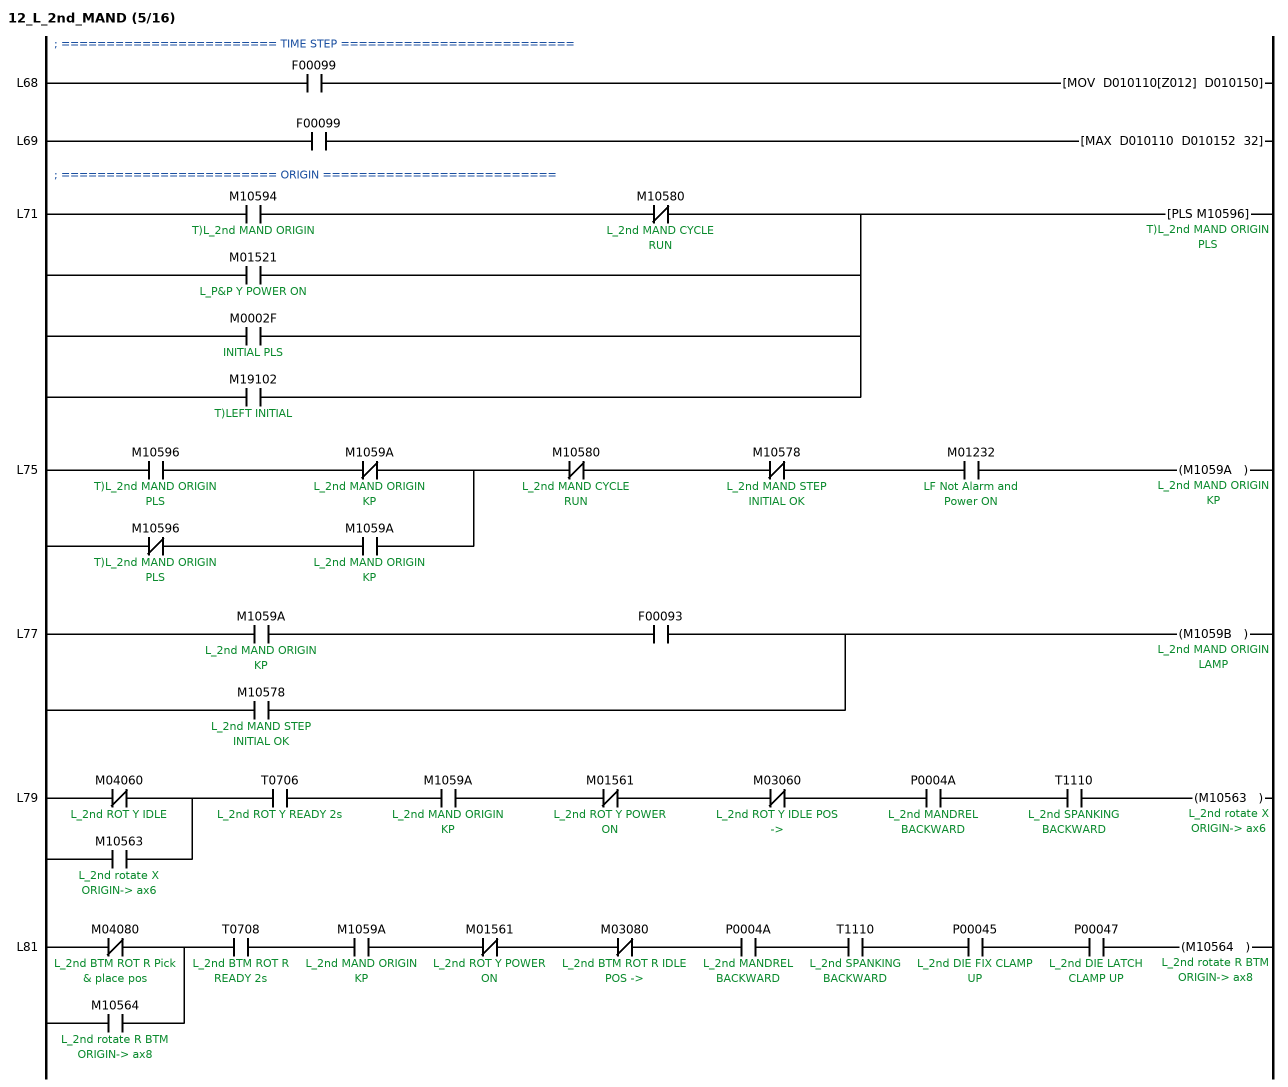
[picture p72: 12_L_2nd_MAND rungs L68-L81]
// ======================== TIME STEP ==========================
; L68
LOAD      F00099
MOV       D010110[Z012] D010150
; L69
LOAD      F00099
MAX       D010110 D010152 32
// ======================== ORIGIN ==========================
; L71
LOAD      M10594	// T)L_2nd MAND ORIGIN
AND NOT   M10580	// L_2nd MAND CYCLE RUN
OR        M01521	// L_P&P Y POWER ON
OR        M0002F	// INITIAL PLS
OR        M19102	// T)LEFT INITIAL
OUTP      M10596	// T)L_2nd MAND ORIGIN PLS
; L75
LOAD      M10596	// T)L_2nd MAND ORIGIN PLS
AND NOT   M1059A	// L_2nd MAND ORIGIN KP
LOAD NOT  M10596	// T)L_2nd MAND ORIGIN PLS
AND       M1059A	// L_2nd MAND ORIGIN KP
OR LOAD
AND NOT   M10580	// L_2nd MAND CYCLE RUN
AND NOT   M10578	// L_2nd MAND STEP INITIAL OK
AND       M01232	// LF Not Alarm and Power ON
OUT       M1059A	// L_2nd MAND ORIGIN KP
; L77
LOAD      M1059A	// L_2nd MAND ORIGIN KP
AND       F00093
OR        M10578	// L_2nd MAND STEP INITIAL OK
OUT       M1059B	// L_2nd MAND ORIGIN LAMP
; L79
LOAD NOT  M04060	// L_2nd ROT Y IDLE
OR        M10563	// L_2nd rotate X ORIGIN-> ax6
AND       T0706	// L_2nd ROT Y READY 2s
AND       M1059A	// L_2nd MAND ORIGIN KP
AND NOT   M01561	// L_2nd ROT Y POWER ON
AND NOT   M03060	// L_2nd ROT Y IDLE POS ->
AND       P0004A	// L_2nd MANDREL BACKWARD
AND       T1110	// L_2nd SPANKING BACKWARD
OUT       M10563	// L_2nd rotate X ORIGIN-> ax6
; L81
LOAD NOT  M04080	// L_2nd BTM ROT R Pick & place pos
OR        M10564	// L_2nd rotate R BTM  ORIGIN-> ax8
AND       T0708	// L_2nd BTM ROT R READY 2s
AND       M1059A	// L_2nd MAND ORIGIN KP
AND NOT   M01561	// L_2nd ROT Y POWER ON
AND NOT   M03080	// L_2nd BTM ROT R IDLE POS ->
AND       P0004A	// L_2nd MANDREL BACKWARD
AND       T1110	// L_2nd SPANKING BACKWARD
AND       P00045	// L_2nd DIE FIX CLAMP UP
AND       P00047	// L_2nd DIE LATCH CLAMP UP
OUT       M10564	// L_2nd rotate R BTM  ORIGIN-> ax8

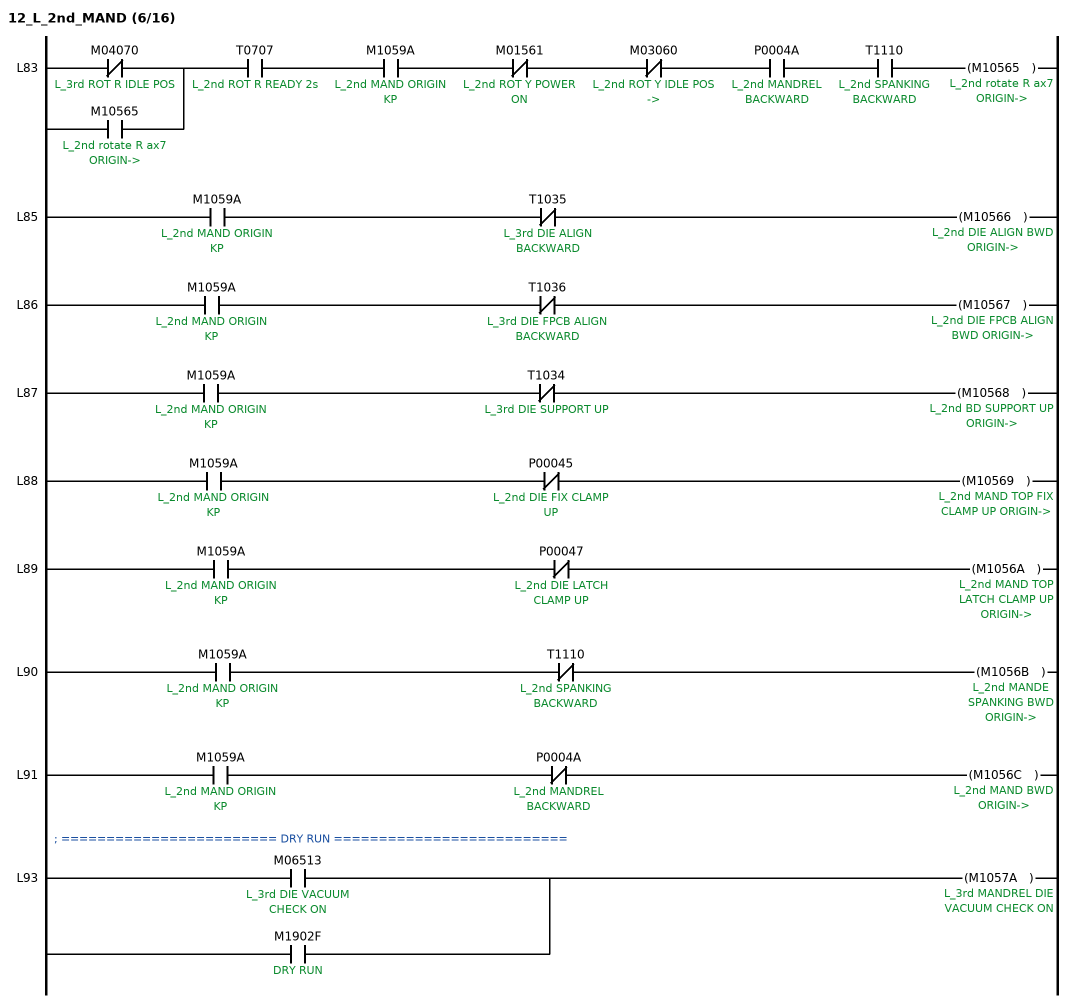
; L83
LOAD NOT  M04070	// L_3rd ROT R IDLE POS
OR        M10565	// L_2nd rotate R ax7 ORIGIN->
AND       T0707	// L_2nd ROT R READY 2s
AND       M1059A	// L_2nd MAND ORIGIN KP
AND NOT   M01561	// L_2nd ROT Y POWER ON
AND NOT   M03060	// L_2nd ROT Y IDLE POS ->
AND       P0004A	// L_2nd MANDREL BACKWARD
AND       T1110	// L_2nd SPANKING BACKWARD
OUT       M10565	// L_2nd rotate R ax7 ORIGIN->
; L85
LOAD      M1059A	// L_2nd MAND ORIGIN KP
AND NOT   T1035	// L_3rd DIE ALIGN BACKWARD
OUT       M10566	// L_2nd DIE ALIGN BWD ORIGIN->
; L86
LOAD      M1059A	// L_2nd MAND ORIGIN KP
AND NOT   T1036	// L_3rd DIE FPCB ALIGN BACKWARD
OUT       M10567	// L_2nd DIE FPCB ALIGN BWD ORIGIN->
; L87
LOAD      M1059A	// L_2nd MAND ORIGIN KP
AND NOT   T1034	// L_3rd DIE SUPPORT UP
OUT       M10568	// L_2nd BD SUPPORT UP ORIGIN->
; L88
LOAD      M1059A	// L_2nd MAND ORIGIN KP
AND NOT   P00045	// L_2nd DIE FIX CLAMP UP
OUT       M10569	// L_2nd MAND TOP FIX CLAMP UP ORIGIN->
; L89
LOAD      M1059A	// L_2nd MAND ORIGIN KP
AND NOT   P00047	// L_2nd DIE LATCH CLAMP UP
OUT       M1056A	// L_2nd MAND TOP LATCH CLAMP UP ORIGIN->
; L90
LOAD      M1059A	// L_2nd MAND ORIGIN KP
AND NOT   T1110	// L_2nd SPANKING BACKWARD
OUT       M1056B	// L_2nd MANDE SPANKING BWD ORIGIN->
; L91
LOAD      M1059A	// L_2nd MAND ORIGIN KP
AND NOT   P0004A	// L_2nd MANDREL BACKWARD
OUT       M1056C	// L_2nd MAND BWD ORIGIN->
// ======================== DRY RUN ==========================
; L93
LOAD      M06513	// L_3rd DIE VACUUM CHECK ON
OR        M1902F	// DRY RUN
OUT       M1057A	// L_3rd MANDREL DIE VACUUM CHECK ON

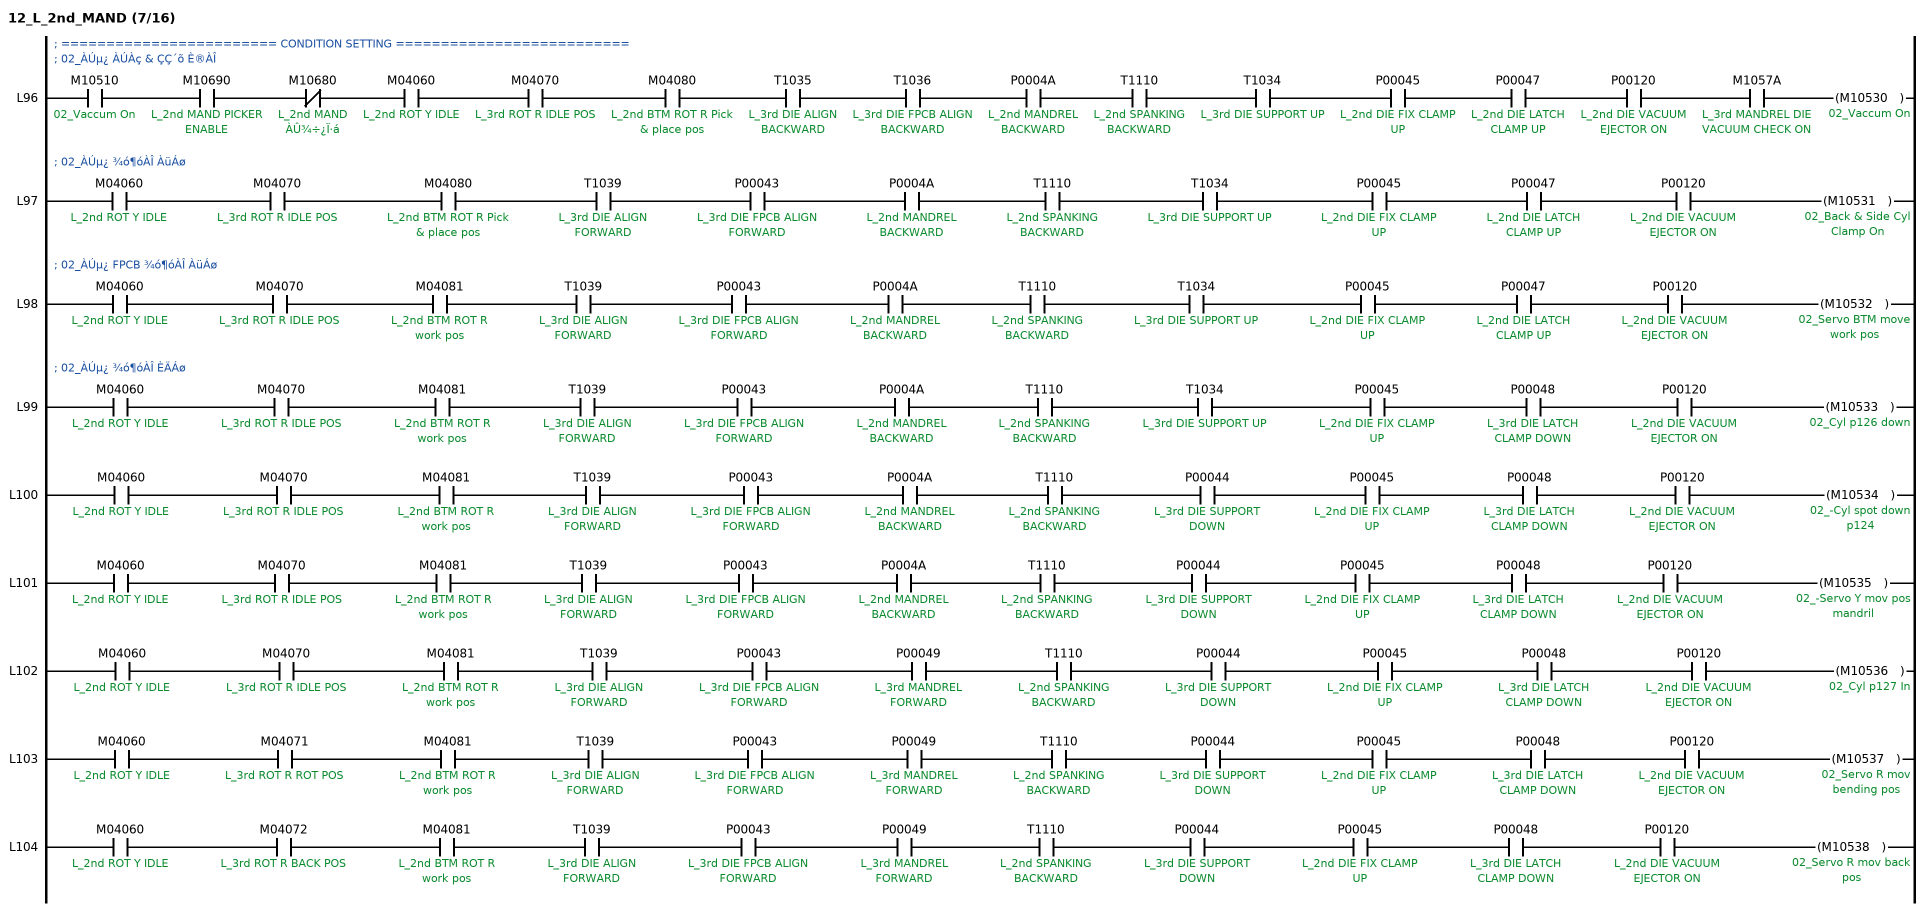
// ======================== CONDITION SETTING ==========================
; L96
LOAD      M10510	// 02_Vaccum On
AND       M10690	// L_2nd MAND PICKER ENABLE
AND NOT   M10680	// L_2nd MAND ÀÛ¾÷¿Ï·á
AND       M04060	// L_2nd ROT Y IDLE
AND       M04070	// L_3rd ROT R IDLE POS
AND       M04080	// L_2nd BTM ROT R Pick & place pos
AND       T1035	// L_3rd DIE ALIGN BACKWARD
AND       T1036	// L_3rd DIE FPCB ALIGN BACKWARD
AND       P0004A	// L_2nd MANDREL BACKWARD
AND       T1110	// L_2nd SPANKING BACKWARD
AND       T1034	// L_3rd DIE SUPPORT UP
AND       P00045	// L_2nd DIE FIX CLAMP UP
AND       P00047	// L_2nd DIE LATCH CLAMP UP
AND       P00120	// L_2nd DIE VACUUM EJECTOR ON
AND       M1057A	// L_3rd MANDREL DIE VACUUM CHECK ON
OUT       M10530	// 02_Vaccum On
// output comment: 02_ÀÚµ¿ ÀÚÀç & ÇÇ´õ È®ÀÎ
; L97
LOAD      M04060	// L_2nd ROT Y IDLE
AND       M04070	// L_3rd ROT R IDLE POS
AND       M04080	// L_2nd BTM ROT R Pick & place pos
AND       T1039	// L_3rd DIE ALIGN FORWARD
AND       P00043	// L_3rd DIE FPCB ALIGN FORWARD
AND       P0004A	// L_2nd MANDREL BACKWARD
AND       T1110	// L_2nd SPANKING BACKWARD
AND       T1034	// L_3rd DIE SUPPORT UP
AND       P00045	// L_2nd DIE FIX CLAMP UP
AND       P00047	// L_2nd DIE LATCH CLAMP UP
AND       P00120	// L_2nd DIE VACUUM EJECTOR ON
OUT       M10531	// 02_Back & Side Cyl Clamp On
// output comment: 02_ÀÚµ¿ ¾ó¶óÀÎ ÀüÁø
; L98
LOAD      M04060	// L_2nd ROT Y IDLE
AND       M04070	// L_3rd ROT R IDLE POS
AND       M04081	// L_2nd BTM ROT R work pos
AND       T1039	// L_3rd DIE ALIGN FORWARD
AND       P00043	// L_3rd DIE FPCB ALIGN FORWARD
AND       P0004A	// L_2nd MANDREL BACKWARD
AND       T1110	// L_2nd SPANKING BACKWARD
AND       T1034	// L_3rd DIE SUPPORT UP
AND       P00045	// L_2nd DIE FIX CLAMP UP
AND       P00047	// L_2nd DIE LATCH CLAMP UP
AND       P00120	// L_2nd DIE VACUUM EJECTOR ON
OUT       M10532	// 02_Servo BTM move work pos
// output comment: 02_ÀÚµ¿ FPCB ¾ó¶óÀÎ ÀüÁø
; L99
LOAD      M04060	// L_2nd ROT Y IDLE
AND       M04070	// L_3rd ROT R IDLE POS
AND       M04081	// L_2nd BTM ROT R work pos
AND       T1039	// L_3rd DIE ALIGN FORWARD
AND       P00043	// L_3rd DIE FPCB ALIGN FORWARD
AND       P0004A	// L_2nd MANDREL BACKWARD
AND       T1110	// L_2nd SPANKING BACKWARD
AND       T1034	// L_3rd DIE SUPPORT UP
AND       P00045	// L_2nd DIE FIX CLAMP UP
AND       P00048	// L_3rd DIE LATCH CLAMP DOWN
AND       P00120	// L_2nd DIE VACUUM EJECTOR ON
OUT       M10533	// 02_Cyl p126 down
// output comment: 02_ÀÚµ¿ ¾ó¶óÀÎ ÈÄÁø
; L100
LOAD      M04060	// L_2nd ROT Y IDLE
AND       M04070	// L_3rd ROT R IDLE POS
AND       M04081	// L_2nd BTM ROT R work pos
AND       T1039	// L_3rd DIE ALIGN FORWARD
AND       P00043	// L_3rd DIE FPCB ALIGN FORWARD
AND       P0004A	// L_2nd MANDREL BACKWARD
AND       T1110	// L_2nd SPANKING BACKWARD
AND       P00044	// L_3rd DIE SUPPORT DOWN
AND       P00045	// L_2nd DIE FIX CLAMP UP
AND       P00048	// L_3rd DIE LATCH CLAMP DOWN
AND       P00120	// L_2nd DIE VACUUM EJECTOR ON
OUT       M10534	// 02_-Cyl spot down p124
; L101
LOAD      M04060	// L_2nd ROT Y IDLE
AND       M04070	// L_3rd ROT R IDLE POS
AND       M04081	// L_2nd BTM ROT R work pos
AND       T1039	// L_3rd DIE ALIGN FORWARD
AND       P00043	// L_3rd DIE FPCB ALIGN FORWARD
AND       P0004A	// L_2nd MANDREL BACKWARD
AND       T1110	// L_2nd SPANKING BACKWARD
AND       P00044	// L_3rd DIE SUPPORT DOWN
AND       P00045	// L_2nd DIE FIX CLAMP UP
AND       P00048	// L_3rd DIE LATCH CLAMP DOWN
AND       P00120	// L_2nd DIE VACUUM EJECTOR ON
OUT       M10535	// 02_-Servo Y mov pos mandril
; L102
LOAD      M04060	// L_2nd ROT Y IDLE
AND       M04070	// L_3rd ROT R IDLE POS
AND       M04081	// L_2nd BTM ROT R work pos
AND       T1039	// L_3rd DIE ALIGN FORWARD
AND       P00043	// L_3rd DIE FPCB ALIGN FORWARD
AND       P00049	// L_3rd MANDREL FORWARD
AND       T1110	// L_2nd SPANKING BACKWARD
AND       P00044	// L_3rd DIE SUPPORT DOWN
AND       P00045	// L_2nd DIE FIX CLAMP UP
AND       P00048	// L_3rd DIE LATCH CLAMP DOWN
AND       P00120	// L_2nd DIE VACUUM EJECTOR ON
OUT       M10536	// 02_Cyl p127 In
; L103
LOAD      M04060	// L_2nd ROT Y IDLE
AND       M04071	// L_3rd ROT R ROT POS
AND       M04081	// L_2nd BTM ROT R work pos
AND       T1039	// L_3rd DIE ALIGN FORWARD
AND       P00043	// L_3rd DIE FPCB ALIGN FORWARD
AND       P00049	// L_3rd MANDREL FORWARD
AND       T1110	// L_2nd SPANKING BACKWARD
AND       P00044	// L_3rd DIE SUPPORT DOWN
AND       P00045	// L_2nd DIE FIX CLAMP UP
AND       P00048	// L_3rd DIE LATCH CLAMP DOWN
AND       P00120	// L_2nd DIE VACUUM EJECTOR ON
OUT       M10537	// 02_Servo R mov bending pos
; L104
LOAD      M04060	// L_2nd ROT Y IDLE
AND       M04072	// L_3rd ROT R BACK POS
AND       M04081	// L_2nd BTM ROT R work pos
AND       T1039	// L_3rd DIE ALIGN FORWARD
AND       P00043	// L_3rd DIE FPCB ALIGN FORWARD
AND       P00049	// L_3rd MANDREL FORWARD
AND       T1110	// L_2nd SPANKING BACKWARD
AND       P00044	// L_3rd DIE SUPPORT DOWN
AND       P00045	// L_2nd DIE FIX CLAMP UP
AND       P00048	// L_3rd DIE LATCH CLAMP DOWN
AND       P00120	// L_2nd DIE VACUUM EJECTOR ON
OUT       M10538	// 02_Servo R mov back pos

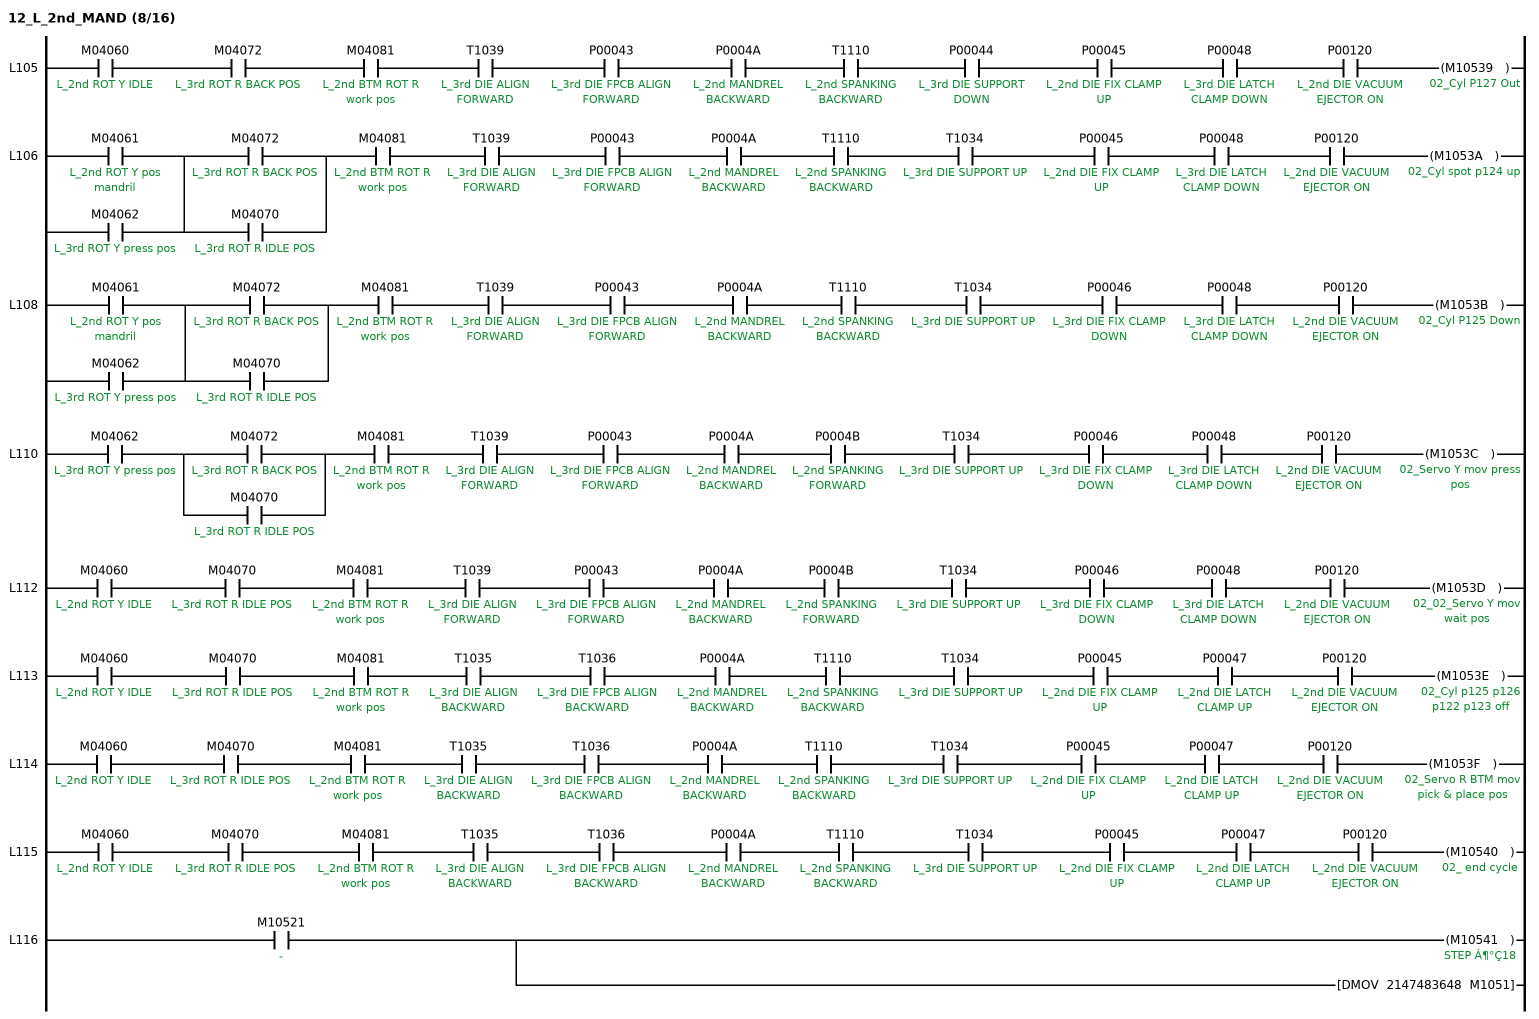
; L105
LOAD      M04060	// L_2nd ROT Y IDLE
AND       M04072	// L_3rd ROT R BACK POS
AND       M04081	// L_2nd BTM ROT R work pos
AND       T1039	// L_3rd DIE ALIGN FORWARD
AND       P00043	// L_3rd DIE FPCB ALIGN FORWARD
AND       P0004A	// L_2nd MANDREL BACKWARD
AND       T1110	// L_2nd SPANKING BACKWARD
AND       P00044	// L_3rd DIE SUPPORT DOWN
AND       P00045	// L_2nd DIE FIX CLAMP UP
AND       P00048	// L_3rd DIE LATCH CLAMP DOWN
AND       P00120	// L_2nd DIE VACUUM EJECTOR ON
OUT       M10539	// 02_Cyl P127 Out
; L106
LOAD      M04061	// L_2nd ROT Y pos mandril
OR        M04062	// L_3rd ROT Y press pos
LOAD      M04072	// L_3rd ROT R BACK POS
OR        M04070	// L_3rd ROT R IDLE POS
AND LOAD
AND       M04081	// L_2nd BTM ROT R work pos
AND       T1039	// L_3rd DIE ALIGN FORWARD
AND       P00043	// L_3rd DIE FPCB ALIGN FORWARD
AND       P0004A	// L_2nd MANDREL BACKWARD
AND       T1110	// L_2nd SPANKING BACKWARD
AND       T1034	// L_3rd DIE SUPPORT UP
AND       P00045	// L_2nd DIE FIX CLAMP UP
AND       P00048	// L_3rd DIE LATCH CLAMP DOWN
AND       P00120	// L_2nd DIE VACUUM EJECTOR ON
OUT       M1053A	// 02_Cyl spot p124 up
; L108
LOAD      M04061	// L_2nd ROT Y pos mandril
OR        M04062	// L_3rd ROT Y press pos
LOAD      M04072	// L_3rd ROT R BACK POS
OR        M04070	// L_3rd ROT R IDLE POS
AND LOAD
AND       M04081	// L_2nd BTM ROT R work pos
AND       T1039	// L_3rd DIE ALIGN FORWARD
AND       P00043	// L_3rd DIE FPCB ALIGN FORWARD
AND       P0004A	// L_2nd MANDREL BACKWARD
AND       T1110	// L_2nd SPANKING BACKWARD
AND       T1034	// L_3rd DIE SUPPORT UP
AND       P00046	// L_3rd DIE FIX CLAMP DOWN
AND       P00048	// L_3rd DIE LATCH CLAMP DOWN
AND       P00120	// L_2nd DIE VACUUM EJECTOR ON
OUT       M1053B	// 02_Cyl P125 Down
; L110
LOAD      M04062	// L_3rd ROT Y press pos
LOAD      M04072	// L_3rd ROT R BACK POS
OR        M04070	// L_3rd ROT R IDLE POS
AND LOAD
AND       M04081	// L_2nd BTM ROT R work pos
AND       T1039	// L_3rd DIE ALIGN FORWARD
AND       P00043	// L_3rd DIE FPCB ALIGN FORWARD
AND       P0004A	// L_2nd MANDREL BACKWARD
AND       P0004B	// L_2nd SPANKING FORWARD
AND       T1034	// L_3rd DIE SUPPORT UP
AND       P00046	// L_3rd DIE FIX CLAMP DOWN
AND       P00048	// L_3rd DIE LATCH CLAMP DOWN
AND       P00120	// L_2nd DIE VACUUM EJECTOR ON
OUT       M1053C	// 02_Servo Y mov press pos
; L112
LOAD      M04060	// L_2nd ROT Y IDLE
AND       M04070	// L_3rd ROT R IDLE POS
AND       M04081	// L_2nd BTM ROT R work pos
AND       T1039	// L_3rd DIE ALIGN FORWARD
AND       P00043	// L_3rd DIE FPCB ALIGN FORWARD
AND       P0004A	// L_2nd MANDREL BACKWARD
AND       P0004B	// L_2nd SPANKING FORWARD
AND       T1034	// L_3rd DIE SUPPORT UP
AND       P00046	// L_3rd DIE FIX CLAMP DOWN
AND       P00048	// L_3rd DIE LATCH CLAMP DOWN
AND       P00120	// L_2nd DIE VACUUM EJECTOR ON
OUT       M1053D	// 02_02_Servo Y mov wait pos
; L113
LOAD      M04060	// L_2nd ROT Y IDLE
AND       M04070	// L_3rd ROT R IDLE POS
AND       M04081	// L_2nd BTM ROT R work pos
AND       T1035	// L_3rd DIE ALIGN BACKWARD
AND       T1036	// L_3rd DIE FPCB ALIGN BACKWARD
AND       P0004A	// L_2nd MANDREL BACKWARD
AND       T1110	// L_2nd SPANKING BACKWARD
AND       T1034	// L_3rd DIE SUPPORT UP
AND       P00045	// L_2nd DIE FIX CLAMP UP
AND       P00047	// L_2nd DIE LATCH CLAMP UP
AND       P00120	// L_2nd DIE VACUUM EJECTOR ON
OUT       M1053E	// 02_Cyl p125 p126 p122 p123 off
; L114
LOAD      M04060	// L_2nd ROT Y IDLE
AND       M04070	// L_3rd ROT R IDLE POS
AND       M04081	// L_2nd BTM ROT R work pos
AND       T1035	// L_3rd DIE ALIGN BACKWARD
AND       T1036	// L_3rd DIE FPCB ALIGN BACKWARD
AND       P0004A	// L_2nd MANDREL BACKWARD
AND       T1110	// L_2nd SPANKING BACKWARD
AND       T1034	// L_3rd DIE SUPPORT UP
AND       P00045	// L_2nd DIE FIX CLAMP UP
AND       P00047	// L_2nd DIE LATCH CLAMP UP
AND       P00120	// L_2nd DIE VACUUM EJECTOR ON
OUT       M1053F	// 02_Servo R BTM mov pick & place pos
; L115
LOAD      M04060	// L_2nd ROT Y IDLE
AND       M04070	// L_3rd ROT R IDLE POS
AND       M04081	// L_2nd BTM ROT R work pos
AND       T1035	// L_3rd DIE ALIGN BACKWARD
AND       T1036	// L_3rd DIE FPCB ALIGN BACKWARD
AND       P0004A	// L_2nd MANDREL BACKWARD
AND       T1110	// L_2nd SPANKING BACKWARD
AND       T1034	// L_3rd DIE SUPPORT UP
AND       P00045	// L_2nd DIE FIX CLAMP UP
AND       P00047	// L_2nd DIE LATCH CLAMP UP
AND       P00120	// L_2nd DIE VACUUM EJECTOR ON
OUT       M10540	// 02_ end cycle
; L116
LOAD      M10521	// -
OUT       M10541	// STEP Á¶°Ç18
DMOV      2147483648 M1051

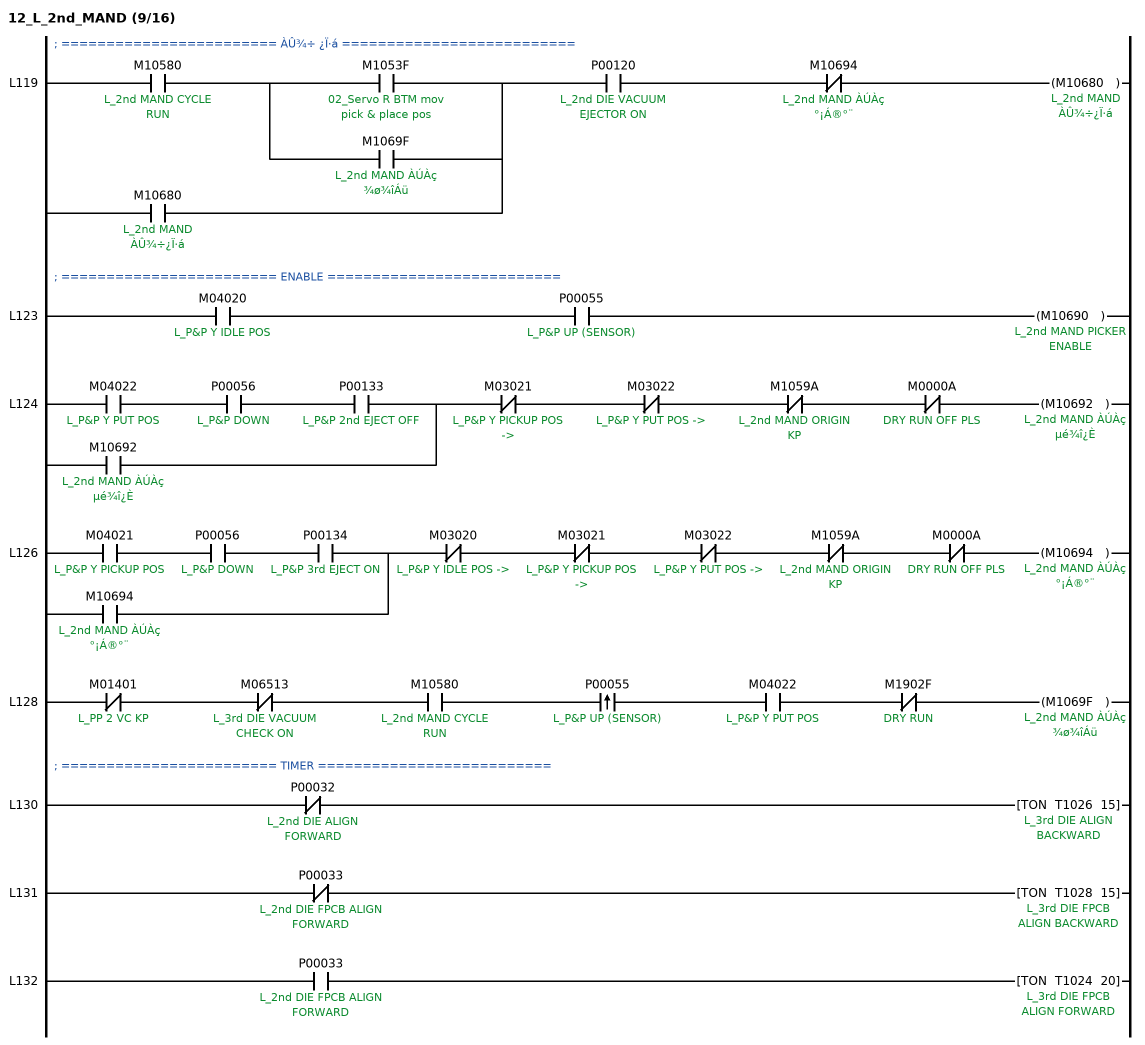
// ======================== ÀÛ¾÷ ¿Ï·á ==========================
; L119
LOAD      M10580	// L_2nd MAND CYCLE RUN
LOAD      M1053F	// 02_Servo R BTM mov pick & place pos
OR        M1069F	// L_2nd MAND ÀÚÀç ¾ø¾îÁü
AND LOAD
OR        M10680	// L_2nd MAND ÀÛ¾÷¿Ï·á
AND       P00120	// L_2nd DIE VACUUM EJECTOR ON
AND NOT   M10694	// L_2nd MAND ÀÚÀç °¡Á®°¨
OUT       M10680	// L_2nd MAND ÀÛ¾÷¿Ï·á
// ======================== ENABLE ==========================
; L123
LOAD      M04020	// L_P&P Y IDLE POS
AND       P00055	// L_P&P UP (SENSOR)
OUT       M10690	// L_2nd MAND PICKER ENABLE
; L124
LOAD      M04022	// L_P&P Y PUT POS
AND       P00056	// L_P&P DOWN
AND       P00133	// L_P&P 2nd EJECT OFF
OR        M10692	// L_2nd MAND ÀÚÀç µé¾î¿È
AND NOT   M03021	// L_P&P Y PICKUP POS ->
AND NOT   M03022	// L_P&P Y PUT POS ->
AND NOT   M1059A	// L_2nd MAND ORIGIN KP
AND NOT   M0000A	// DRY RUN OFF PLS
OUT       M10692	// L_2nd MAND ÀÚÀç µé¾î¿È
; L126
LOAD      M04021	// L_P&P Y PICKUP POS
AND       P00056	// L_P&P DOWN
AND       P00134	// L_P&P 3rd EJECT ON
OR        M10694	// L_2nd MAND ÀÚÀç °¡Á®°¨
AND NOT   M03020	// L_P&P Y IDLE POS ->
AND NOT   M03021	// L_P&P Y PICKUP POS ->
AND NOT   M03022	// L_P&P Y PUT POS ->
AND NOT   M1059A	// L_2nd MAND ORIGIN KP
AND NOT   M0000A	// DRY RUN OFF PLS
OUT       M10694	// L_2nd MAND ÀÚÀç °¡Á®°¨
; L128
LOAD NOT  M01401	// L_PP 2 VC KP
AND NOT   M06513	// L_3rd DIE VACUUM CHECK ON
AND       M10580	// L_2nd MAND CYCLE RUN
ANDP      P00055	// L_P&P UP (SENSOR)
AND       M04022	// L_P&P Y PUT POS
AND NOT   M1902F	// DRY RUN
OUT       M1069F	// L_2nd MAND ÀÚÀç ¾ø¾îÁü
// ======================== TIMER ==========================
; L130
LOAD NOT  P00032	// L_2nd DIE ALIGN FORWARD
TON       T1026 15	// L_3rd DIE ALIGN BACKWARD
; L131
LOAD NOT  P00033	// L_2nd DIE FPCB ALIGN FORWARD
TON       T1028 15	// L_3rd DIE FPCB ALIGN BACKWARD
; L132
LOAD      P00033	// L_2nd DIE FPCB ALIGN FORWARD
TON       T1024 20	// L_3rd DIE FPCB ALIGN FORWARD

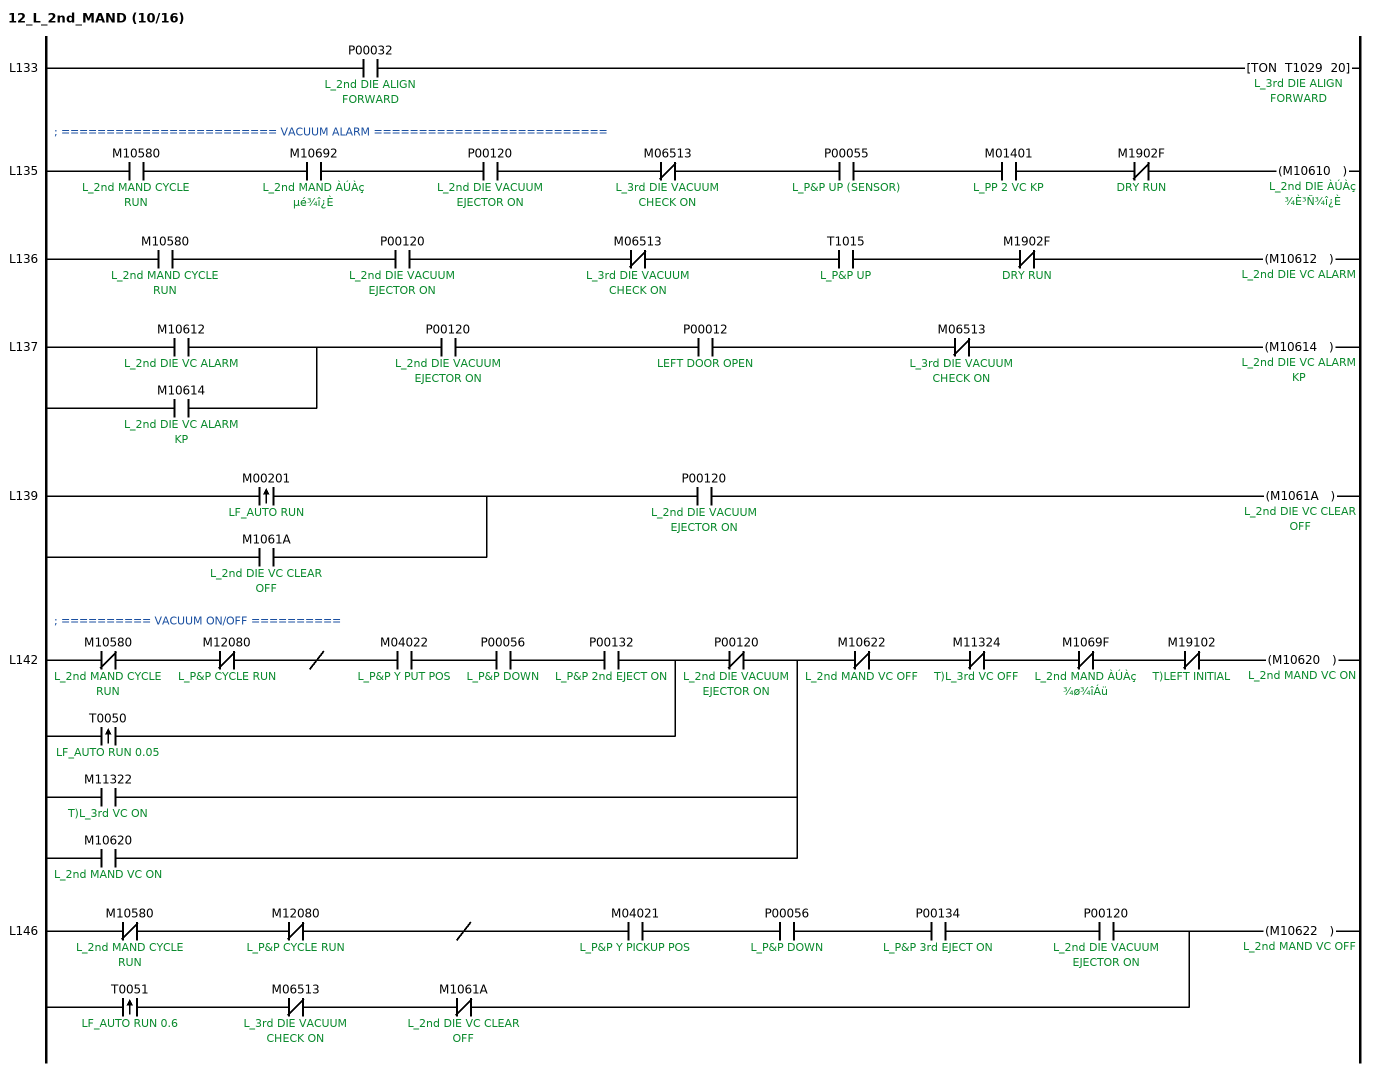
; L133
LOAD      P00032	// L_2nd DIE ALIGN FORWARD
TON       T1029 20	// L_3rd DIE ALIGN FORWARD
// ======================== VACUUM ALARM ==========================
; L135
LOAD      M10580	// L_2nd MAND CYCLE RUN
AND       M10692	// L_2nd MAND ÀÚÀç µé¾î¿È
AND       P00120	// L_2nd DIE VACUUM EJECTOR ON
AND NOT   M06513	// L_3rd DIE VACUUM CHECK ON
AND       P00055	// L_P&P UP (SENSOR)
AND       M01401	// L_PP 2 VC KP
AND NOT   M1902F	// DRY RUN
OUT       M10610	// L_2nd DIE ÀÚÀç ¾È³Ñ¾î¿È
; L136
LOAD      M10580	// L_2nd MAND CYCLE RUN
AND       P00120	// L_2nd DIE VACUUM EJECTOR ON
AND NOT   M06513	// L_3rd DIE VACUUM CHECK ON
AND       T1015	// L_P&P UP
AND NOT   M1902F	// DRY RUN
OUT       M10612	// L_2nd DIE VC ALARM
; L137
LOAD      M10612	// L_2nd DIE VC ALARM
OR        M10614	// L_2nd DIE VC ALARM KP
AND       P00120	// L_2nd DIE VACUUM EJECTOR ON
AND       P00012	// LEFT DOOR OPEN
AND NOT   M06513	// L_3rd DIE VACUUM CHECK ON
OUT       M10614	// L_2nd DIE VC ALARM KP
; L139
LOADP     M00201	// LF_AUTO RUN
OR        M1061A	// L_2nd DIE VC CLEAR OFF
AND       P00120	// L_2nd DIE VACUUM EJECTOR ON
OUT       M1061A	// L_2nd DIE VC CLEAR OFF
// ========== VACUUM ON/OFF ==========
; L142
LOAD NOT  M10580	// L_2nd MAND CYCLE RUN
AND NOT   M12080	// L_P&P CYCLE RUN
NOT
AND       M04022	// L_P&P Y PUT POS
AND       P00056	// L_P&P DOWN
AND       P00132	// L_P&P 2nd EJECT ON
ORP       T0050	// LF_AUTO RUN 0.05
AND NOT   P00120	// L_2nd DIE VACUUM EJECTOR ON
OR        M11322	// T)L_3rd VC ON
OR        M10620	// L_2nd MAND VC ON
AND NOT   M10622	// L_2nd MAND VC OFF
AND NOT   M11324	// T)L_3rd VC OFF
AND NOT   M1069F	// L_2nd MAND ÀÚÀç ¾ø¾îÁü
AND NOT   M19102	// T)LEFT INITIAL
OUT       M10620	// L_2nd MAND VC ON
; L146
LOAD NOT  M10580	// L_2nd MAND CYCLE RUN
AND NOT   M12080	// L_P&P CYCLE RUN
NOT
AND       M04021	// L_P&P Y PICKUP POS
AND       P00056	// L_P&P DOWN
AND       P00134	// L_P&P 3rd EJECT ON
AND       P00120	// L_2nd DIE VACUUM EJECTOR ON
LOADP     T0051	// LF_AUTO RUN 0.6
AND NOT   M06513	// L_3rd DIE VACUUM CHECK ON
AND NOT   M1061A	// L_2nd DIE VC CLEAR OFF
OR LOAD
OUT       M10622	// L_2nd MAND VC OFF

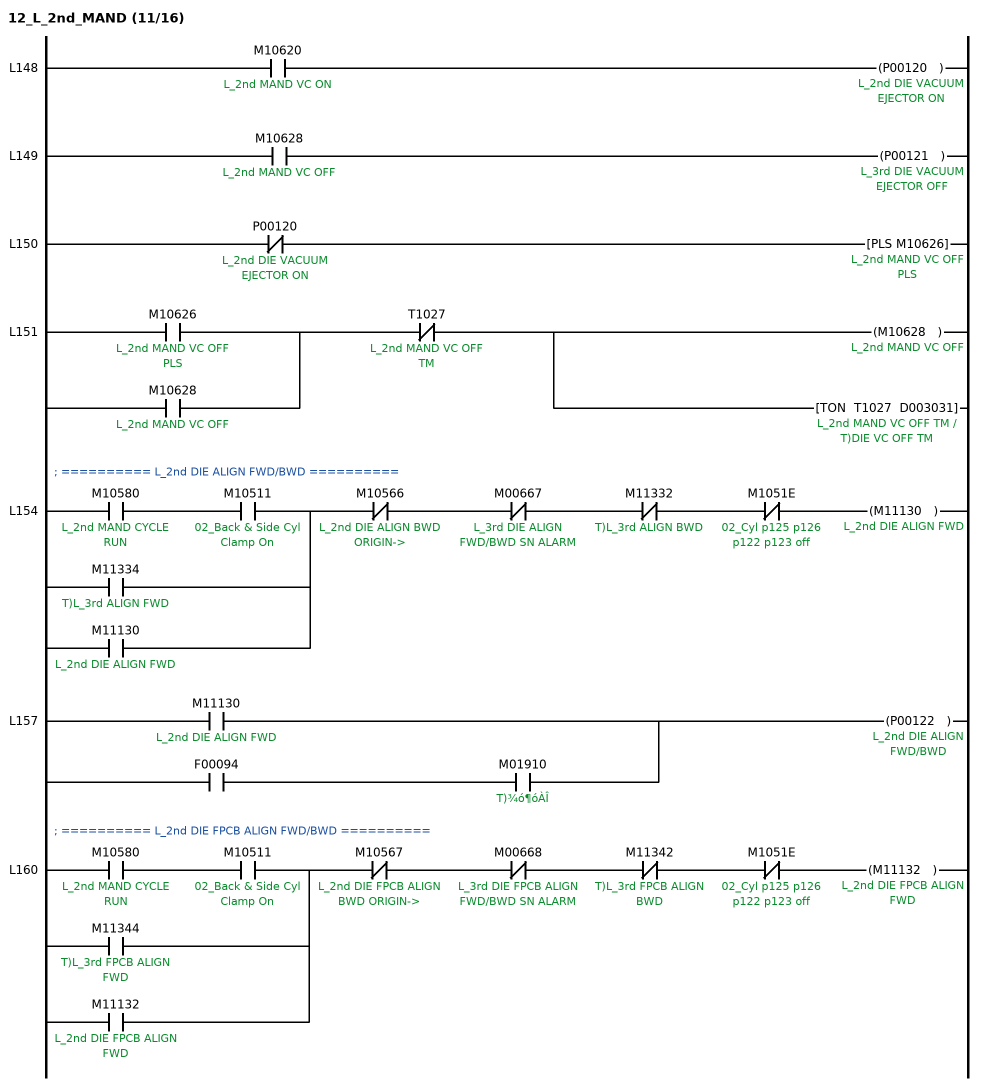
; L148
LOAD      M10620	// L_2nd MAND VC ON
OUT       P00120	// L_2nd DIE VACUUM EJECTOR ON
; L149
LOAD      M10628	// L_2nd MAND VC OFF
OUT       P00121	// L_3rd DIE VACUUM EJECTOR OFF
; L150
LOAD NOT  P00120	// L_2nd DIE VACUUM EJECTOR ON
OUTP      M10626	// L_2nd MAND VC OFF PLS
; L151
LOAD      M10626	// L_2nd MAND VC OFF PLS
OR        M10628	// L_2nd MAND VC OFF
AND NOT   T1027	// L_2nd MAND VC OFF TM
OUT       M10628	// L_2nd MAND VC OFF
TON       T1027 D003031	// L_2nd MAND VC OFF TM / T)DIE VC OFF TM
// ========== L_2nd DIE ALIGN FWD/BWD ==========
; L154
LOAD      M10580	// L_2nd MAND CYCLE RUN
AND       M10511	// 02_Back & Side Cyl Clamp On
OR        M11334	// T)L_3rd ALIGN FWD
OR        M11130	// L_2nd DIE ALIGN FWD
AND NOT   M10566	// L_2nd DIE ALIGN BWD ORIGIN->
AND NOT   M00667	// L_3rd DIE ALIGN FWD/BWD SN ALARM
AND NOT   M11332	// T)L_3rd ALIGN BWD
AND NOT   M1051E	// 02_Cyl p125 p126 p122 p123 off
OUT       M11130	// L_2nd DIE ALIGN FWD
; L157
LOAD      M11130	// L_2nd DIE ALIGN FWD
LOAD      F00094
AND       M01910	// T)¾ó¶óÀÎ
OR LOAD
OUT       P00122	// L_2nd DIE ALIGN FWD/BWD
// ========== L_2nd DIE FPCB ALIGN FWD/BWD ==========
; L160
LOAD      M10580	// L_2nd MAND CYCLE RUN
AND       M10511	// 02_Back & Side Cyl Clamp On
OR        M11344	// T)L_3rd FPCB ALIGN FWD
OR        M11132	// L_2nd DIE FPCB ALIGN FWD
AND NOT   M10567	// L_2nd DIE FPCB ALIGN BWD ORIGIN->
AND NOT   M00668	// L_3rd DIE FPCB ALIGN FWD/BWD SN ALARM
AND NOT   M11342	// T)L_3rd FPCB ALIGN BWD
AND NOT   M1051E	// 02_Cyl p125 p126 p122 p123 off
OUT       M11132	// L_2nd DIE FPCB ALIGN FWD

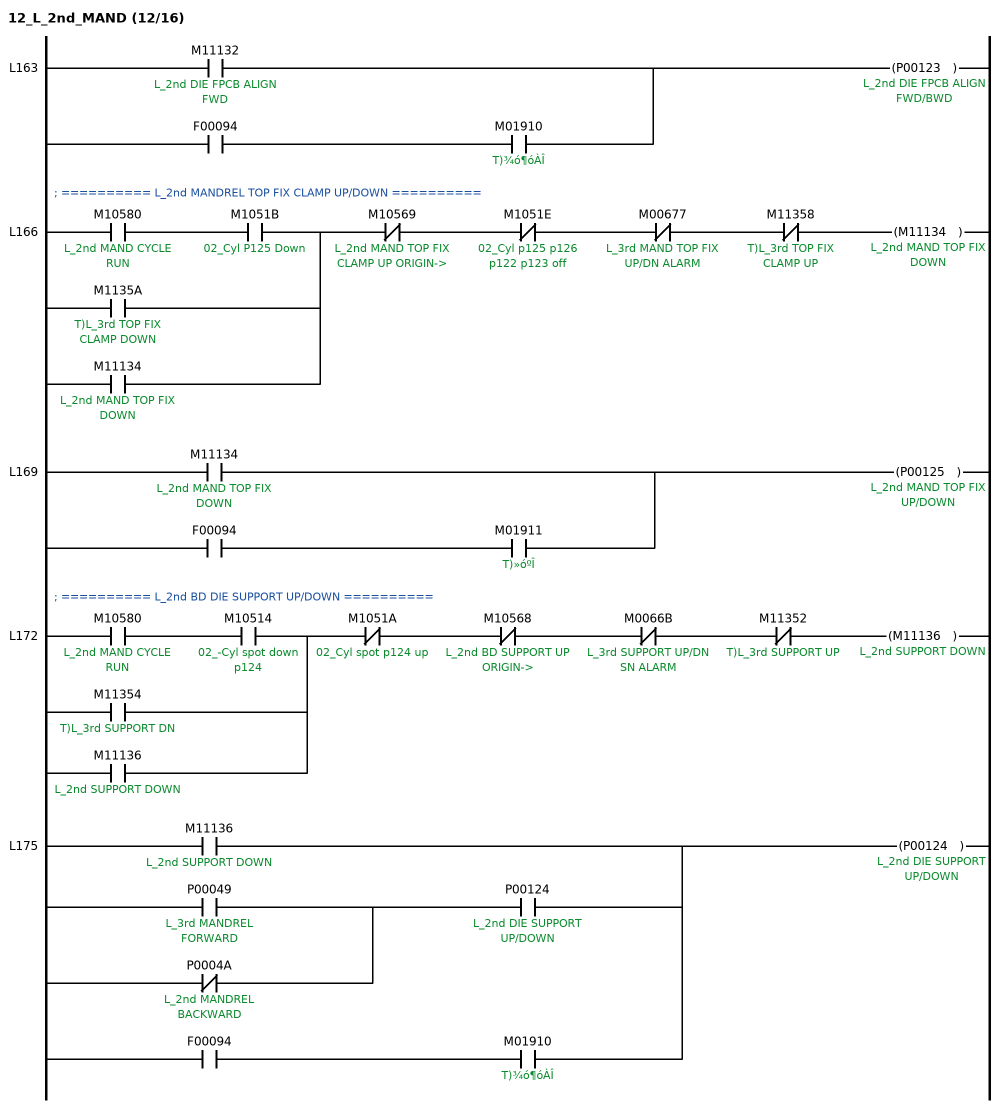
; L163
LOAD      M11132	// L_2nd DIE FPCB ALIGN FWD
LOAD      F00094
AND       M01910	// T)¾ó¶óÀÎ
OR LOAD
OUT       P00123	// L_2nd DIE FPCB ALIGN FWD/BWD
// ========== L_2nd MANDREL TOP FIX CLAMP UP/DOWN ==========
; L166
LOAD      M10580	// L_2nd MAND CYCLE RUN
AND       M1051B	// 02_Cyl P125 Down
OR        M1135A	// T)L_3rd TOP FIX CLAMP DOWN
OR        M11134	// L_2nd MAND TOP FIX DOWN
AND NOT   M10569	// L_2nd MAND TOP FIX CLAMP UP ORIGIN->
AND NOT   M1051E	// 02_Cyl p125 p126 p122 p123 off
AND NOT   M00677	// L_3rd MAND TOP FIX UP/DN ALARM
AND NOT   M11358	// T)L_3rd TOP FIX CLAMP UP
OUT       M11134	// L_2nd MAND TOP FIX DOWN
; L169
LOAD      M11134	// L_2nd MAND TOP FIX DOWN
LOAD      F00094
AND       M01911	// T)»óºÎ
OR LOAD
OUT       P00125	// L_2nd MAND TOP FIX UP/DOWN
// ========== L_2nd BD DIE SUPPORT UP/DOWN ==========
; L172
LOAD      M10580	// L_2nd MAND CYCLE RUN
AND       M10514	// 02_-Cyl spot down p124
OR        M11354	// T)L_3rd SUPPORT DN
OR        M11136	// L_2nd SUPPORT DOWN
AND NOT   M1051A	// 02_Cyl spot p124 up
AND NOT   M10568	// L_2nd BD SUPPORT UP ORIGIN->
AND NOT   M0066B	// L_3rd SUPPORT UP/DN SN ALARM
AND NOT   M11352	// T)L_3rd SUPPORT UP
OUT       M11136	// L_2nd SUPPORT DOWN
; L175
LOAD      M11136	// L_2nd SUPPORT DOWN
LOAD      P00049	// L_3rd MANDREL FORWARD
OR NOT    P0004A	// L_2nd MANDREL BACKWARD
AND       P00124	// L_2nd DIE SUPPORT UP/DOWN
OR LOAD
LOAD      F00094
AND       M01910	// T)¾ó¶óÀÎ
OR LOAD
OUT       P00124	// L_2nd DIE SUPPORT UP/DOWN

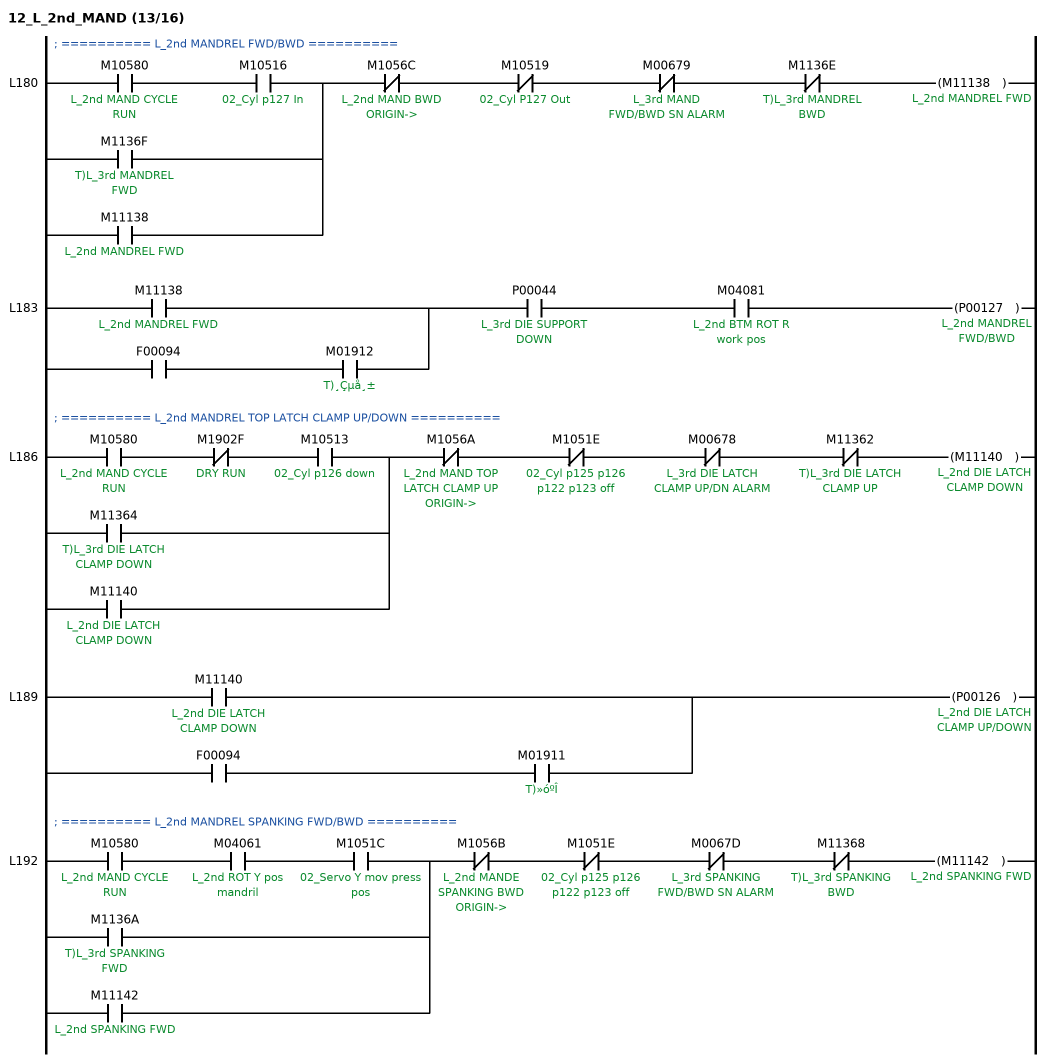
// ========== L_2nd MANDREL FWD/BWD ==========
; L180
LOAD      M10580	// L_2nd MAND CYCLE RUN
AND       M10516	// 02_Cyl p127 In
OR        M1136F	// T)L_3rd MANDREL FWD
OR        M11138	// L_2nd MANDREL FWD
AND NOT   M1056C	// L_2nd MAND BWD ORIGIN->
AND NOT   M10519	// 02_Cyl P127 Out
AND NOT   M00679	// L_3rd MAND FWD/BWD SN ALARM
AND NOT   M1136E	// T)L_3rd MANDREL BWD
OUT       M11138	// L_2nd MANDREL FWD
; L183
LOAD      M11138	// L_2nd MANDREL FWD
LOAD      F00094
AND       M01912	// T)¸Çµå¸±
OR LOAD
AND       P00044	// L_3rd DIE SUPPORT DOWN
AND       M04081	// L_2nd BTM ROT R work pos
OUT       P00127	// L_2nd MANDREL FWD/BWD
// ========== L_2nd MANDREL TOP LATCH CLAMP UP/DOWN ==========
; L186
LOAD      M10580	// L_2nd MAND CYCLE RUN
AND NOT   M1902F	// DRY RUN
AND       M10513	// 02_Cyl p126 down
OR        M11364	// T)L_3rd DIE LATCH CLAMP DOWN
OR        M11140	// L_2nd DIE LATCH CLAMP DOWN
AND NOT   M1056A	// L_2nd MAND TOP LATCH CLAMP UP ORIGIN->
AND NOT   M1051E	// 02_Cyl p125 p126 p122 p123 off
AND NOT   M00678	// L_3rd DIE LATCH CLAMP UP/DN ALARM
AND NOT   M11362	// T)L_3rd DIE LATCH CLAMP UP
OUT       M11140	// L_2nd DIE LATCH CLAMP DOWN
; L189
LOAD      M11140	// L_2nd DIE LATCH CLAMP DOWN
LOAD      F00094
AND       M01911	// T)»óºÎ
OR LOAD
OUT       P00126	// L_2nd DIE LATCH CLAMP UP/DOWN
// ========== L_2nd MANDREL SPANKING FWD/BWD ==========
; L192
LOAD      M10580	// L_2nd MAND CYCLE RUN
AND       M04061	// L_2nd ROT Y pos mandril
AND       M1051C	// 02_Servo Y mov press pos
OR        M1136A	// T)L_3rd SPANKING FWD
OR        M11142	// L_2nd SPANKING FWD
AND NOT   M1056B	// L_2nd MANDE SPANKING BWD ORIGIN->
AND NOT   M1051E	// 02_Cyl p125 p126 p122 p123 off
AND NOT   M0067D	// L_3rd SPANKING FWD/BWD SN ALARM
AND NOT   M11368	// T)L_3rd SPANKING BWD
OUT       M11142	// L_2nd SPANKING FWD

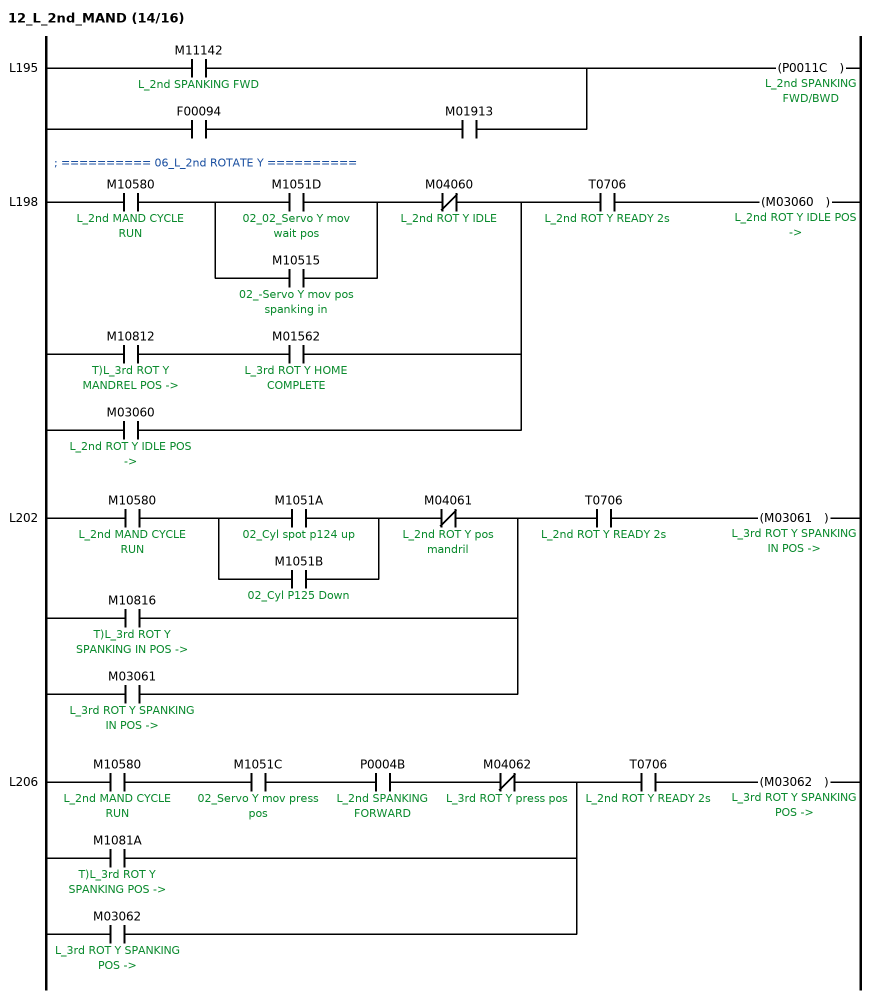
; L195
LOAD      M11142	// L_2nd SPANKING FWD
LOAD      F00094
AND       M01913
OR LOAD
OUT       P0011C	// L_2nd SPANKING FWD/BWD
// ========== 06_L_2nd ROTATE Y ==========
; L198
LOAD      M10580	// L_2nd MAND CYCLE RUN
LOAD      M1051D	// 02_02_Servo Y mov wait pos
OR        M10515	// 02_-Servo Y mov pos spanking in
AND LOAD
AND NOT   M04060	// L_2nd ROT Y IDLE
LOAD      M10812	// T)L_3rd ROT Y MANDREL POS ->
AND       M01562	// L_3rd ROT Y HOME COMPLETE
OR LOAD
OR        M03060	// L_2nd ROT Y IDLE POS ->
AND       T0706	// L_2nd ROT Y READY 2s
OUT       M03060	// L_2nd ROT Y IDLE POS ->
; L202
LOAD      M10580	// L_2nd MAND CYCLE RUN
LOAD      M1051A	// 02_Cyl spot p124 up
OR        M1051B	// 02_Cyl P125 Down
AND LOAD
AND NOT   M04061	// L_2nd ROT Y pos mandril
OR        M10816	// T)L_3rd ROT Y SPANKING IN POS ->
OR        M03061	// L_3rd ROT Y SPANKING IN POS ->
AND       T0706	// L_2nd ROT Y READY 2s
OUT       M03061	// L_3rd ROT Y SPANKING IN POS ->
; L206
LOAD      M10580	// L_2nd MAND CYCLE RUN
AND       M1051C	// 02_Servo Y mov press pos
AND       P0004B	// L_2nd SPANKING FORWARD
AND NOT   M04062	// L_3rd ROT Y press pos
OR        M1081A	// T)L_3rd ROT Y SPANKING POS ->
OR        M03062	// L_3rd ROT Y SPANKING POS ->
AND       T0706	// L_2nd ROT Y READY 2s
OUT       M03062	// L_3rd ROT Y SPANKING POS ->

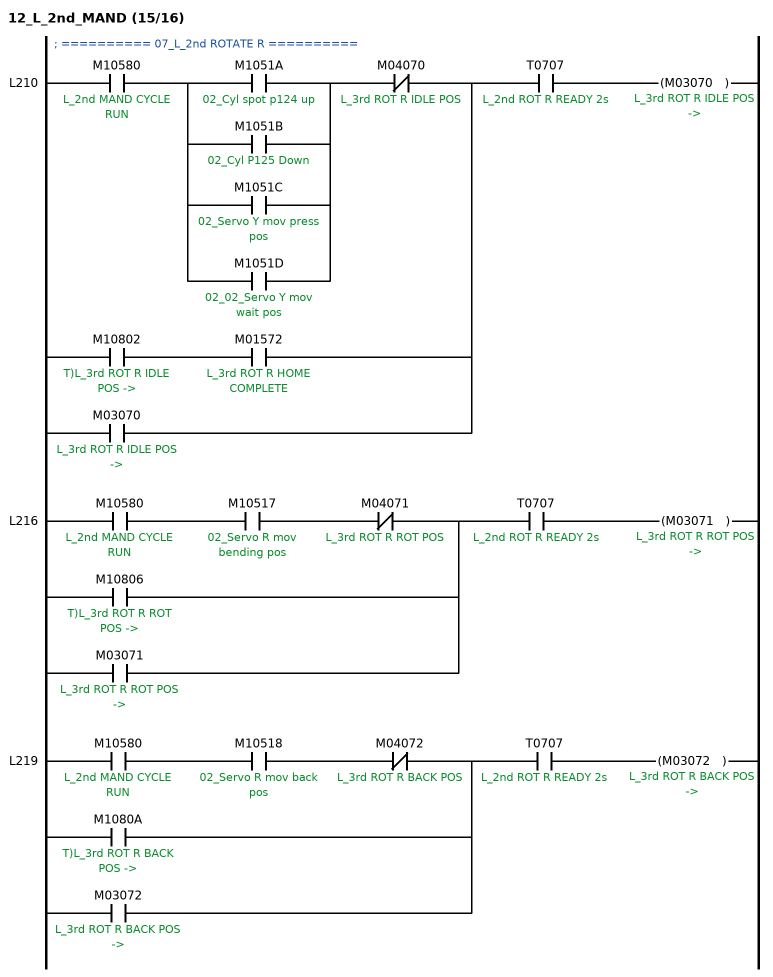
// ========== 07_L_2nd ROTATE R ==========
; L210
LOAD      M10580	// L_2nd MAND CYCLE RUN
LOAD      M1051A	// 02_Cyl spot p124 up
OR        M1051B	// 02_Cyl P125 Down
OR        M1051C	// 02_Servo Y mov press pos
OR        M1051D	// 02_02_Servo Y mov wait pos
AND LOAD
AND NOT   M04070	// L_3rd ROT R IDLE POS
LOAD      M10802	// T)L_3rd ROT R IDLE POS ->
AND       M01572	// L_3rd ROT R HOME COMPLETE
OR LOAD
OR        M03070	// L_3rd ROT R IDLE POS ->
AND       T0707	// L_2nd ROT R READY 2s
OUT       M03070	// L_3rd ROT R IDLE POS ->
; L216
LOAD      M10580	// L_2nd MAND CYCLE RUN
AND       M10517	// 02_Servo R mov bending pos
AND NOT   M04071	// L_3rd ROT R ROT POS
OR        M10806	// T)L_3rd ROT R ROT POS ->
OR        M03071	// L_3rd ROT R ROT POS ->
AND       T0707	// L_2nd ROT R READY 2s
OUT       M03071	// L_3rd ROT R ROT POS ->
; L219
LOAD      M10580	// L_2nd MAND CYCLE RUN
AND       M10518	// 02_Servo R mov back pos
AND NOT   M04072	// L_3rd ROT R BACK POS
OR        M1080A	// T)L_3rd ROT R BACK POS ->
OR        M03072	// L_3rd ROT R BACK POS ->
AND       T0707	// L_2nd ROT R READY 2s
OUT       M03072	// L_3rd ROT R BACK POS ->

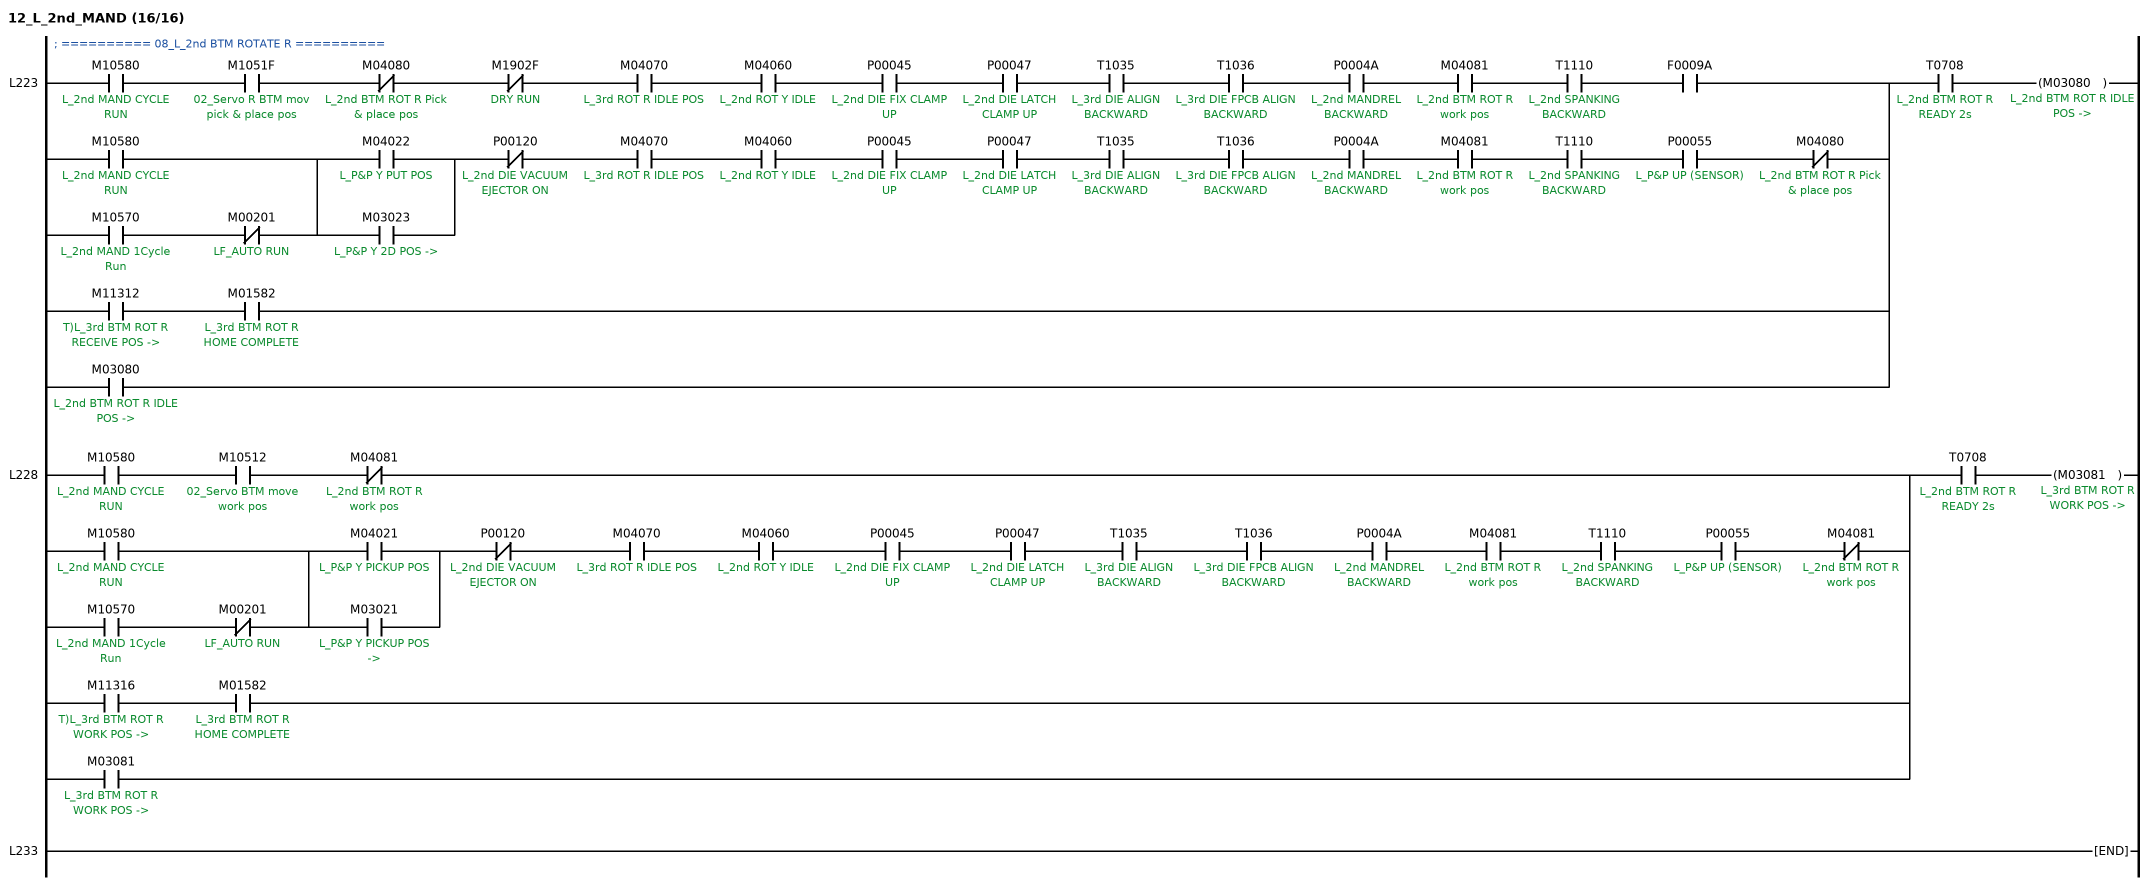
// ========== 08_L_2nd BTM ROTATE R ==========
; L223
LOAD      M10580	// L_2nd MAND CYCLE RUN
AND       M1051F	// 02_Servo R BTM mov pick & place pos
AND NOT   M04080	// L_2nd BTM ROT R Pick & place pos
AND NOT   M1902F	// DRY RUN
AND       M04070	// L_3rd ROT R IDLE POS
AND       M04060	// L_2nd ROT Y IDLE
AND       P00045	// L_2nd DIE FIX CLAMP UP
AND       P00047	// L_2nd DIE LATCH CLAMP UP
AND       T1035	// L_3rd DIE ALIGN BACKWARD
AND       T1036	// L_3rd DIE FPCB ALIGN BACKWARD
AND       P0004A	// L_2nd MANDREL BACKWARD
AND       M04081	// L_2nd BTM ROT R work pos
AND       T1110	// L_2nd SPANKING BACKWARD
AND       F0009A
LOAD      M10580	// L_2nd MAND CYCLE RUN
LOAD      M10570	// L_2nd MAND 1Cycle Run
AND NOT   M00201	// LF_AUTO RUN
OR LOAD
LOAD      M04022	// L_P&P Y PUT POS
OR        M03023	// L_P&P Y 2D POS ->
AND LOAD
AND NOT   P00120	// L_2nd DIE VACUUM EJECTOR ON
AND       M04070	// L_3rd ROT R IDLE POS
AND       M04060	// L_2nd ROT Y IDLE
AND       P00045	// L_2nd DIE FIX CLAMP UP
AND       P00047	// L_2nd DIE LATCH CLAMP UP
AND       T1035	// L_3rd DIE ALIGN BACKWARD
AND       T1036	// L_3rd DIE FPCB ALIGN BACKWARD
AND       P0004A	// L_2nd MANDREL BACKWARD
AND       M04081	// L_2nd BTM ROT R work pos
AND       T1110	// L_2nd SPANKING BACKWARD
AND       P00055	// L_P&P UP (SENSOR)
AND NOT   M04080	// L_2nd BTM ROT R Pick & place pos
OR LOAD
LOAD      M11312	// T)L_3rd BTM ROT R RECEIVE POS ->
AND       M01582	// L_3rd BTM ROT R HOME COMPLETE
OR LOAD
OR        M03080	// L_2nd BTM ROT R IDLE POS ->
AND       T0708	// L_2nd BTM ROT R READY 2s
OUT       M03080	// L_2nd BTM ROT R IDLE POS ->
; L228
LOAD      M10580	// L_2nd MAND CYCLE RUN
AND       M10512	// 02_Servo BTM move work pos
AND NOT   M04081	// L_2nd BTM ROT R work pos
LOAD      M10580	// L_2nd MAND CYCLE RUN
LOAD      M10570	// L_2nd MAND 1Cycle Run
AND NOT   M00201	// LF_AUTO RUN
OR LOAD
LOAD      M04021	// L_P&P Y PICKUP POS
OR        M03021	// L_P&P Y PICKUP POS ->
AND LOAD
AND NOT   P00120	// L_2nd DIE VACUUM EJECTOR ON
AND       M04070	// L_3rd ROT R IDLE POS
AND       M04060	// L_2nd ROT Y IDLE
AND       P00045	// L_2nd DIE FIX CLAMP UP
AND       P00047	// L_2nd DIE LATCH CLAMP UP
AND       T1035	// L_3rd DIE ALIGN BACKWARD
AND       T1036	// L_3rd DIE FPCB ALIGN BACKWARD
AND       P0004A	// L_2nd MANDREL BACKWARD
AND       M04081	// L_2nd BTM ROT R work pos
AND       T1110	// L_2nd SPANKING BACKWARD
AND       P00055	// L_P&P UP (SENSOR)
AND NOT   M04081	// L_2nd BTM ROT R work pos
OR LOAD
LOAD      M11316	// T)L_3rd BTM ROT R WORK POS ->
AND       M01582	// L_3rd BTM ROT R HOME COMPLETE
OR LOAD
OR        M03081	// L_3rd BTM ROT R WORK POS ->
AND       T0708	// L_2nd BTM ROT R READY 2s
OUT       M03081	// L_3rd BTM ROT R WORK POS ->
; L233
END

PROGRAM 13_L_3rd_MAND (task: ½ºÄµ ÇÁ·Î±×·¥)

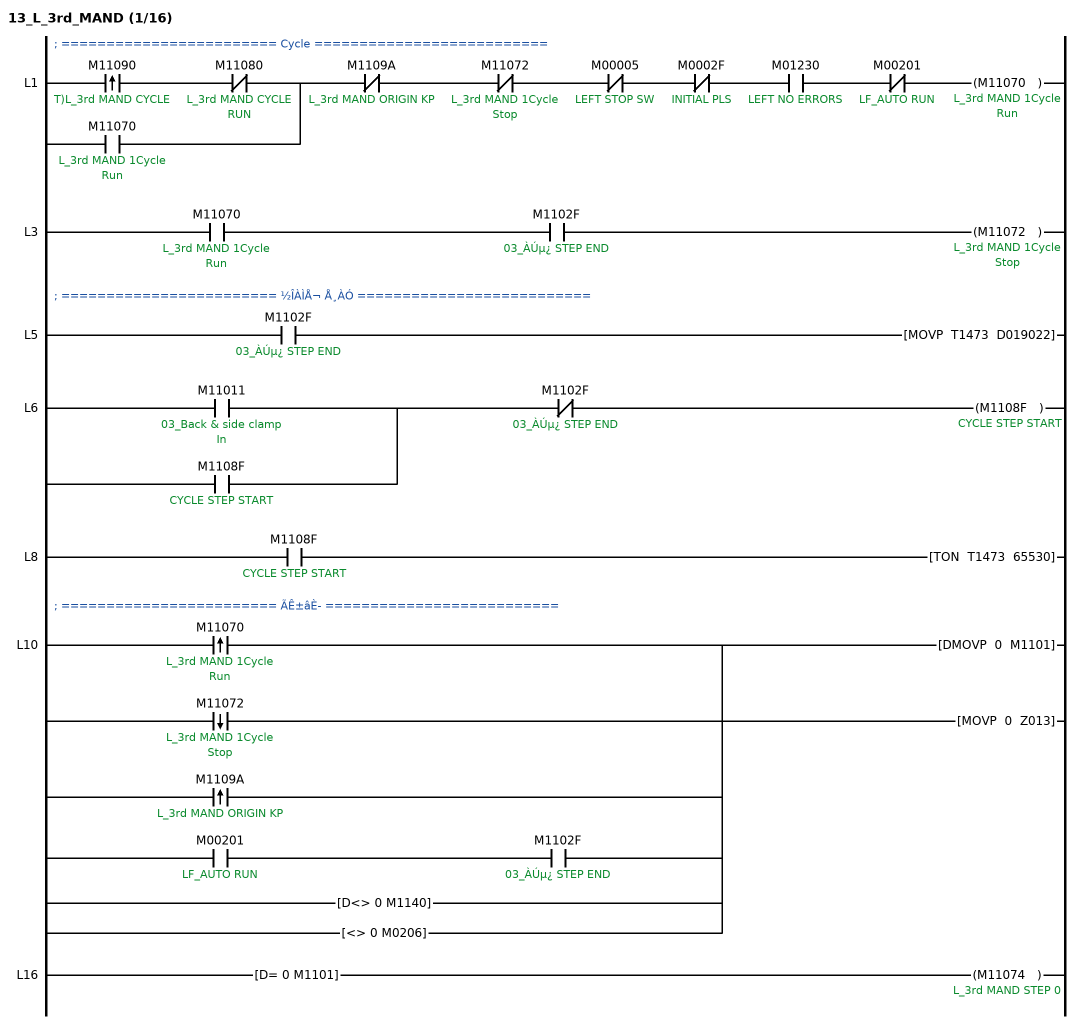
// ======================== Cycle ==========================
; L1
LOADP     M11090	// T)L_3rd MAND CYCLE
AND NOT   M11080	// L_3rd MAND CYCLE RUN
OR        M11070	// L_3rd MAND 1Cycle Run
AND NOT   M1109A	// L_3rd MAND ORIGIN KP
AND NOT   M11072	// L_3rd MAND 1Cycle Stop
AND NOT   M00005	// LEFT STOP SW
AND NOT   M0002F	// INITIAL PLS
AND       M01230	// LEFT NO ERRORS
AND NOT   M00201	// LF_AUTO RUN
OUT       M11070	// L_3rd MAND 1Cycle Run
; L3
LOAD      M11070	// L_3rd MAND 1Cycle Run
AND       M1102F	// 03_ÀÚµ¿ STEP END
OUT       M11072	// L_3rd MAND 1Cycle Stop
// ======================== ½ÎÀÌÅ¬ Å¸ÀÓ ==========================
; L5
LOAD      M1102F	// 03_ÀÚµ¿ STEP END
MOVP      T1473 D019022
; L6
LOAD      M11011	// 03_Back & side clamp In
OR        M1108F	// CYCLE STEP START
AND NOT   M1102F	// 03_ÀÚµ¿ STEP END
OUT       M1108F	// CYCLE STEP START
; L8
LOAD      M1108F	// CYCLE STEP START
TON       T1473 65530
// ======================== ÃÊ±âÈ­ ==========================
; L10
LOADP     M11070	// L_3rd MAND 1Cycle Run
ORN       M11072	// L_3rd MAND 1Cycle Stop
ORP       M1109A	// L_3rd MAND ORIGIN KP
LOAD      M00201	// LF_AUTO RUN
AND       M1102F	// 03_ÀÚµ¿ STEP END
OR LOAD
ORD<>     0 M1140
OR<>      0 M0206
DMOVP     0 M1101
MOVP      0 Z013
; L16
LOADD=    0 M1101
OUT       M11074	// L_3rd MAND STEP 0

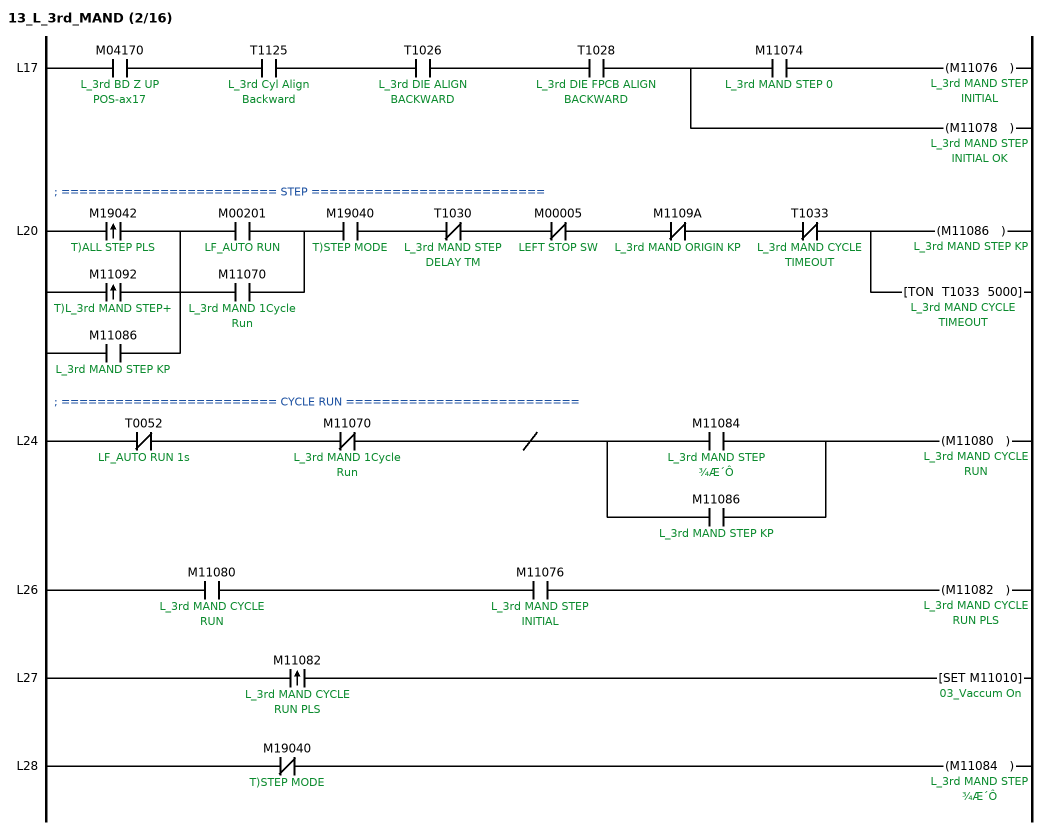
; L17
LOAD      M04170	// L_3rd BD Z UP POS-ax17
AND       T1125	// L_3rd Cyl Align Backward
AND       T1026	// L_3rd DIE ALIGN BACKWARD
AND       T1028	// L_3rd DIE FPCB ALIGN BACKWARD
MPUSH
AND       M11074	// L_3rd MAND STEP 0
OUT       M11076	// L_3rd MAND STEP INITIAL
MPOP
OUT       M11078	// L_3rd MAND STEP INITIAL OK
// ======================== STEP ==========================
; L20
LOADP     M19042	// T)ALL STEP PLS
ORP       M11092	// T)L_3rd MAND STEP+
OR        M11086	// L_3rd MAND STEP KP
LOAD      M00201	// LF_AUTO RUN
OR        M11070	// L_3rd MAND 1Cycle Run
AND LOAD
AND       M19040	// T)STEP MODE
AND NOT   T1030	// L_3rd MAND STEP DELAY TM
AND NOT   M00005	// LEFT STOP SW
AND NOT   M1109A	// L_3rd MAND ORIGIN KP
AND NOT   T1033	// L_3rd MAND CYCLE TIMEOUT
OUT       M11086	// L_3rd MAND STEP KP
TON       T1033 5000	// L_3rd MAND CYCLE TIMEOUT
// ======================== CYCLE RUN ==========================
; L24
LOAD NOT  T0052	// LF_AUTO RUN 1s
AND NOT   M11070	// L_3rd MAND 1Cycle Run
NOT
LOAD      M11084	// L_3rd MAND STEP ¾Æ´Ô
OR        M11086	// L_3rd MAND STEP KP
AND LOAD
OUT       M11080	// L_3rd MAND CYCLE RUN
; L26
LOAD      M11080	// L_3rd MAND CYCLE RUN
AND       M11076	// L_3rd MAND STEP INITIAL
OUT       M11082	// L_3rd MAND CYCLE RUN PLS
; L27
LOADP     M11082	// L_3rd MAND CYCLE RUN PLS
SET       M11010	// 03_Vaccum On
; L28
LOAD NOT  M19040	// T)STEP MODE
OUT       M11084	// L_3rd MAND STEP ¾Æ´Ô

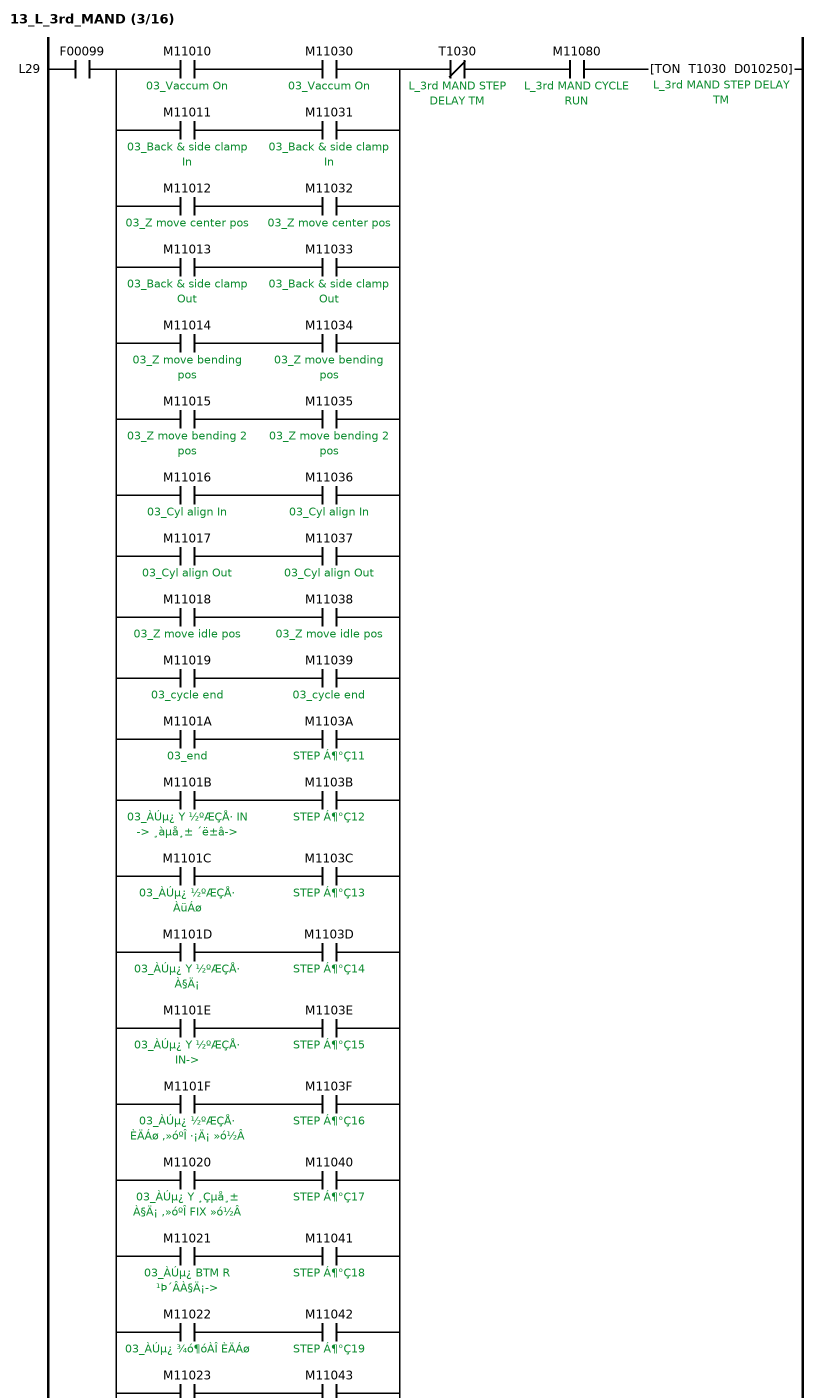

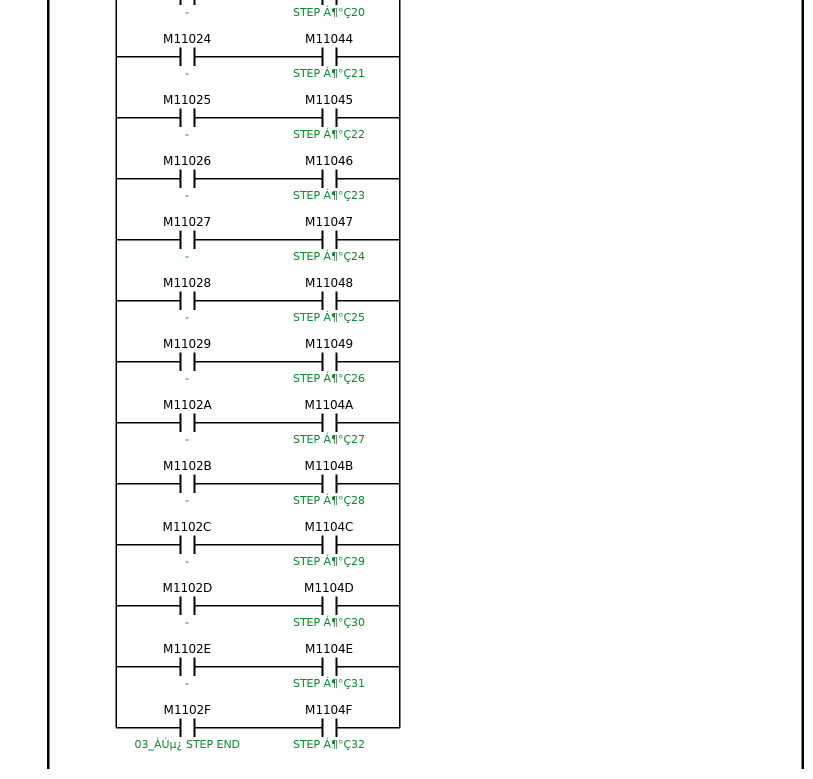
; L29
LOAD      F00099
LOAD      M11010	// 03_Vaccum On
AND       M11030	// 03_Vaccum On
LOAD      M11011	// 03_Back & side clamp In
AND       M11031	// 03_Back & side clamp In
OR LOAD
LOAD      M11012	// 03_Z move center pos
AND       M11032	// 03_Z move center pos
OR LOAD
LOAD      M11013	// 03_Back & side clamp Out
AND       M11033	// 03_Back & side clamp Out
OR LOAD
LOAD      M11014	// 03_Z move bending pos
AND       M11034	// 03_Z move bending pos
OR LOAD
LOAD      M11015	// 03_Z move bending 2 pos
AND       M11035	// 03_Z move bending 2 pos
OR LOAD
LOAD      M11016	// 03_Cyl align In
AND       M11036	// 03_Cyl align In
OR LOAD
LOAD      M11017	// 03_Cyl align Out
AND       M11037	// 03_Cyl align Out
OR LOAD
LOAD      M11018	// 03_Z move idle pos
AND       M11038	// 03_Z move idle pos
OR LOAD
LOAD      M11019	// 03_cycle end
AND       M11039	// 03_cycle end
OR LOAD
LOAD      M1101A	// 03_end
AND       M1103A	// STEP Á¶°Ç11
OR LOAD
LOAD      M1101B	// 03_ÀÚµ¿ Y ½ºÆÇÅ· IN -> ¸àµå¸± ´ë±â->
AND       M1103B	// STEP Á¶°Ç12
OR LOAD
LOAD      M1101C	// 03_ÀÚµ¿ ½ºÆÇÅ· ÀüÁø
AND       M1103C	// STEP Á¶°Ç13
OR LOAD
LOAD      M1101D	// 03_ÀÚµ¿ Y ½ºÆÇÅ· À§Ä¡
AND       M1103D	// STEP Á¶°Ç14
OR LOAD
LOAD      M1101E	// 03_ÀÚµ¿ Y ½ºÆÇÅ· IN->
AND       M1103E	// STEP Á¶°Ç15
OR LOAD
LOAD      M1101F	// 03_ÀÚµ¿ ½ºÆÇÅ· ÈÄÁø ,»óºÎ ·¡Ä¡ »ó½Â
AND       M1103F	// STEP Á¶°Ç16
OR LOAD
LOAD      M11020	// 03_ÀÚµ¿ Y ¸Çµå¸± À§Ä¡ ,»óºÎ FIX »ó½Â
AND       M11040	// STEP Á¶°Ç17
OR LOAD
LOAD      M11021	// 03_ÀÚµ¿ BTM R ¹Þ´ÂÀ§Ä¡->
AND       M11041	// STEP Á¶°Ç18
OR LOAD
LOAD      M11022	// 03_ÀÚµ¿ ¾ó¶óÀÎ ÈÄÁø
AND       M11042	// STEP Á¶°Ç19
OR LOAD
LOAD      M11023	// -
AND       M11043	// STEP Á¶°Ç20
OR LOAD
LOAD      M11024	// -
AND       M11044	// STEP Á¶°Ç21
OR LOAD
LOAD      M11025	// -
AND       M11045	// STEP Á¶°Ç22
OR LOAD
LOAD      M11026	// -
AND       M11046	// STEP Á¶°Ç23
OR LOAD
LOAD      M11027	// -
AND       M11047	// STEP Á¶°Ç24
OR LOAD
LOAD      M11028	// -
AND       M11048	// STEP Á¶°Ç25
OR LOAD
LOAD      M11029	// -
AND       M11049	// STEP Á¶°Ç26
OR LOAD
LOAD      M1102A	// -
AND       M1104A	// STEP Á¶°Ç27
OR LOAD
LOAD      M1102B	// -
AND       M1104B	// STEP Á¶°Ç28
OR LOAD
LOAD      M1102C	// -
AND       M1104C	// STEP Á¶°Ç29
OR LOAD
LOAD      M1102D	// -
AND       M1104D	// STEP Á¶°Ç30
OR LOAD
LOAD      M1102E	// -
AND       M1104E	// STEP Á¶°Ç31
OR LOAD
LOAD      M1102F	// 03_ÀÚµ¿ STEP END
AND       M1104F	// STEP Á¶°Ç32
OR LOAD
AND LOAD
AND NOT   T1030	// L_3rd MAND STEP DELAY TM
AND       M11080	// L_3rd MAND CYCLE RUN
TON       T1030 D010250	// L_3rd MAND STEP DELAY TM

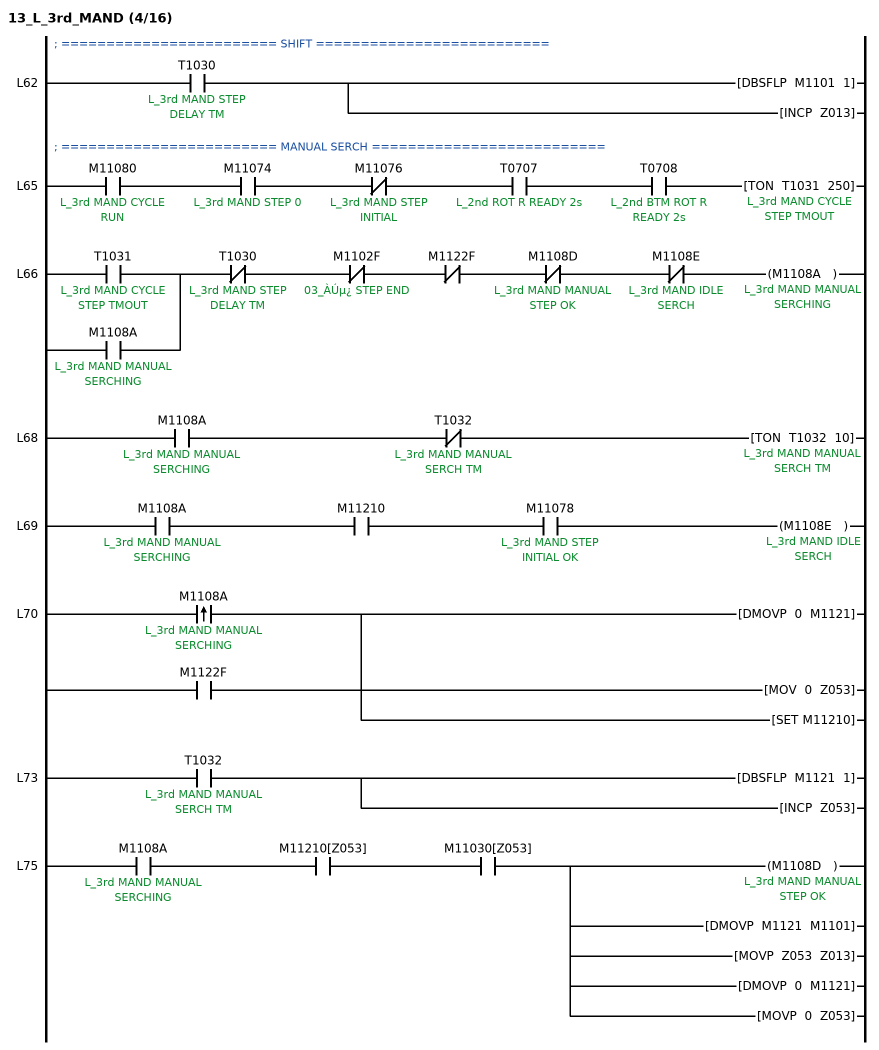
// ======================== SHIFT ==========================
; L62
LOAD      T1030	// L_3rd MAND STEP DELAY TM
DBSFLP    M1101 1
INCP      Z013
// ======================== MANUAL SERCH ==========================
; L65
LOAD      M11080	// L_3rd MAND CYCLE RUN
AND       M11074	// L_3rd MAND STEP 0
AND NOT   M11076	// L_3rd MAND STEP INITIAL
AND       T0707	// L_2nd ROT R READY 2s
AND       T0708	// L_2nd BTM ROT R READY 2s
TON       T1031 250	// L_3rd MAND CYCLE STEP TMOUT
; L66
LOAD      T1031	// L_3rd MAND CYCLE STEP TMOUT
OR        M1108A	// L_3rd MAND MANUAL SERCHING
AND NOT   T1030	// L_3rd MAND STEP DELAY TM
AND NOT   M1102F	// 03_ÀÚµ¿ STEP END
AND NOT   M1122F
AND NOT   M1108D	// L_3rd MAND MANUAL STEP OK
AND NOT   M1108E	// L_3rd MAND IDLE SERCH
OUT       M1108A	// L_3rd MAND MANUAL SERCHING
; L68
LOAD      M1108A	// L_3rd MAND MANUAL SERCHING
AND NOT   T1032	// L_3rd MAND MANUAL SERCH TM
TON       T1032 10	// L_3rd MAND MANUAL SERCH TM
; L69
LOAD      M1108A	// L_3rd MAND MANUAL SERCHING
AND       M11210
AND       M11078	// L_3rd MAND STEP INITIAL OK
OUT       M1108E	// L_3rd MAND IDLE SERCH
; L70
LOADP     M1108A	// L_3rd MAND MANUAL SERCHING
OR        M1122F
DMOVP     0 M1121
MOV       0 Z053
SET       M11210
; L73
LOAD      T1032	// L_3rd MAND MANUAL SERCH TM
DBSFLP    M1121 1
INCP      Z053
; L75
LOAD      M1108A	// L_3rd MAND MANUAL SERCHING
AND       M11210[Z053]
AND       M11030[Z053]
OUT       M1108D	// L_3rd MAND MANUAL STEP OK
DMOVP     M1121 M1101
MOVP      Z053 Z013
DMOVP     0 M1121
MOVP      0 Z053

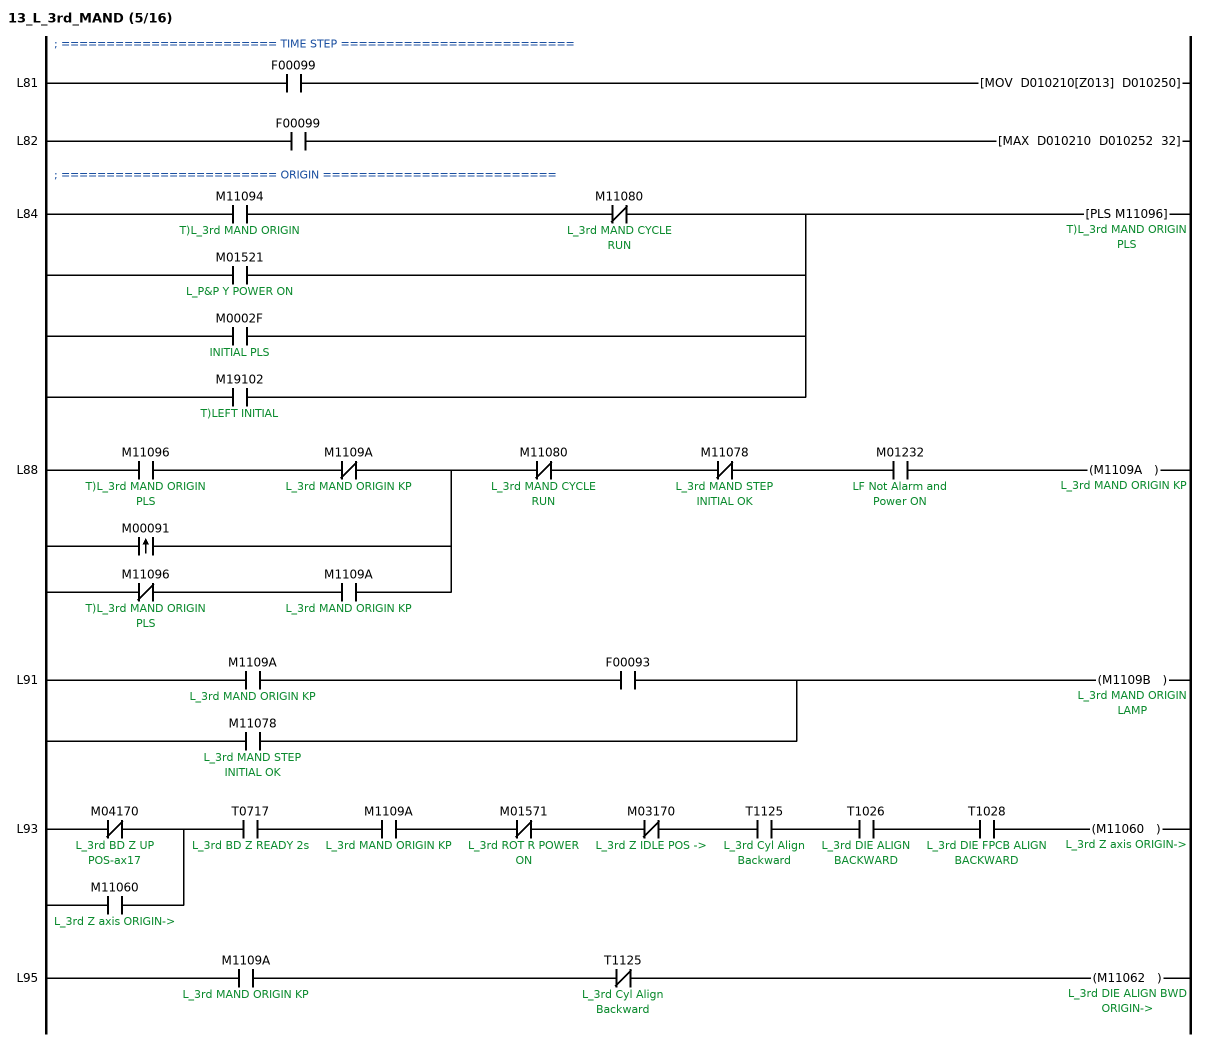
// ======================== TIME STEP ==========================
; L81
LOAD      F00099
MOV       D010210[Z013] D010250
; L82
LOAD      F00099
MAX       D010210 D010252 32
// ======================== ORIGIN ==========================
; L84
LOAD      M11094	// T)L_3rd MAND ORIGIN
AND NOT   M11080	// L_3rd MAND CYCLE RUN
OR        M01521	// L_P&P Y POWER ON
OR        M0002F	// INITIAL PLS
OR        M19102	// T)LEFT INITIAL
OUTP      M11096	// T)L_3rd MAND ORIGIN PLS
; L88
LOAD      M11096	// T)L_3rd MAND ORIGIN PLS
AND NOT   M1109A	// L_3rd MAND ORIGIN KP
ORP       M00091
LOAD NOT  M11096	// T)L_3rd MAND ORIGIN PLS
AND       M1109A	// L_3rd MAND ORIGIN KP
OR LOAD
AND NOT   M11080	// L_3rd MAND CYCLE RUN
AND NOT   M11078	// L_3rd MAND STEP INITIAL OK
AND       M01232	// LF Not Alarm and Power ON
OUT       M1109A	// L_3rd MAND ORIGIN KP
; L91
LOAD      M1109A	// L_3rd MAND ORIGIN KP
AND       F00093
OR        M11078	// L_3rd MAND STEP INITIAL OK
OUT       M1109B	// L_3rd MAND ORIGIN LAMP
; L93
LOAD NOT  M04170	// L_3rd BD Z UP POS-ax17
OR        M11060	// L_3rd Z axis ORIGIN->
AND       T0717	// L_3rd BD Z READY 2s
AND       M1109A	// L_3rd MAND ORIGIN KP
AND NOT   M01571	// L_3rd ROT R POWER ON
AND NOT   M03170	// L_3rd Z IDLE POS ->
AND       T1125	// L_3rd Cyl Align Backward
AND       T1026	// L_3rd DIE ALIGN BACKWARD
AND       T1028	// L_3rd DIE FPCB ALIGN BACKWARD
OUT       M11060	// L_3rd Z axis ORIGIN->
; L95
LOAD      M1109A	// L_3rd MAND ORIGIN KP
AND NOT   T1125	// L_3rd Cyl Align Backward
OUT       M11062	// L_3rd DIE ALIGN BWD ORIGIN->

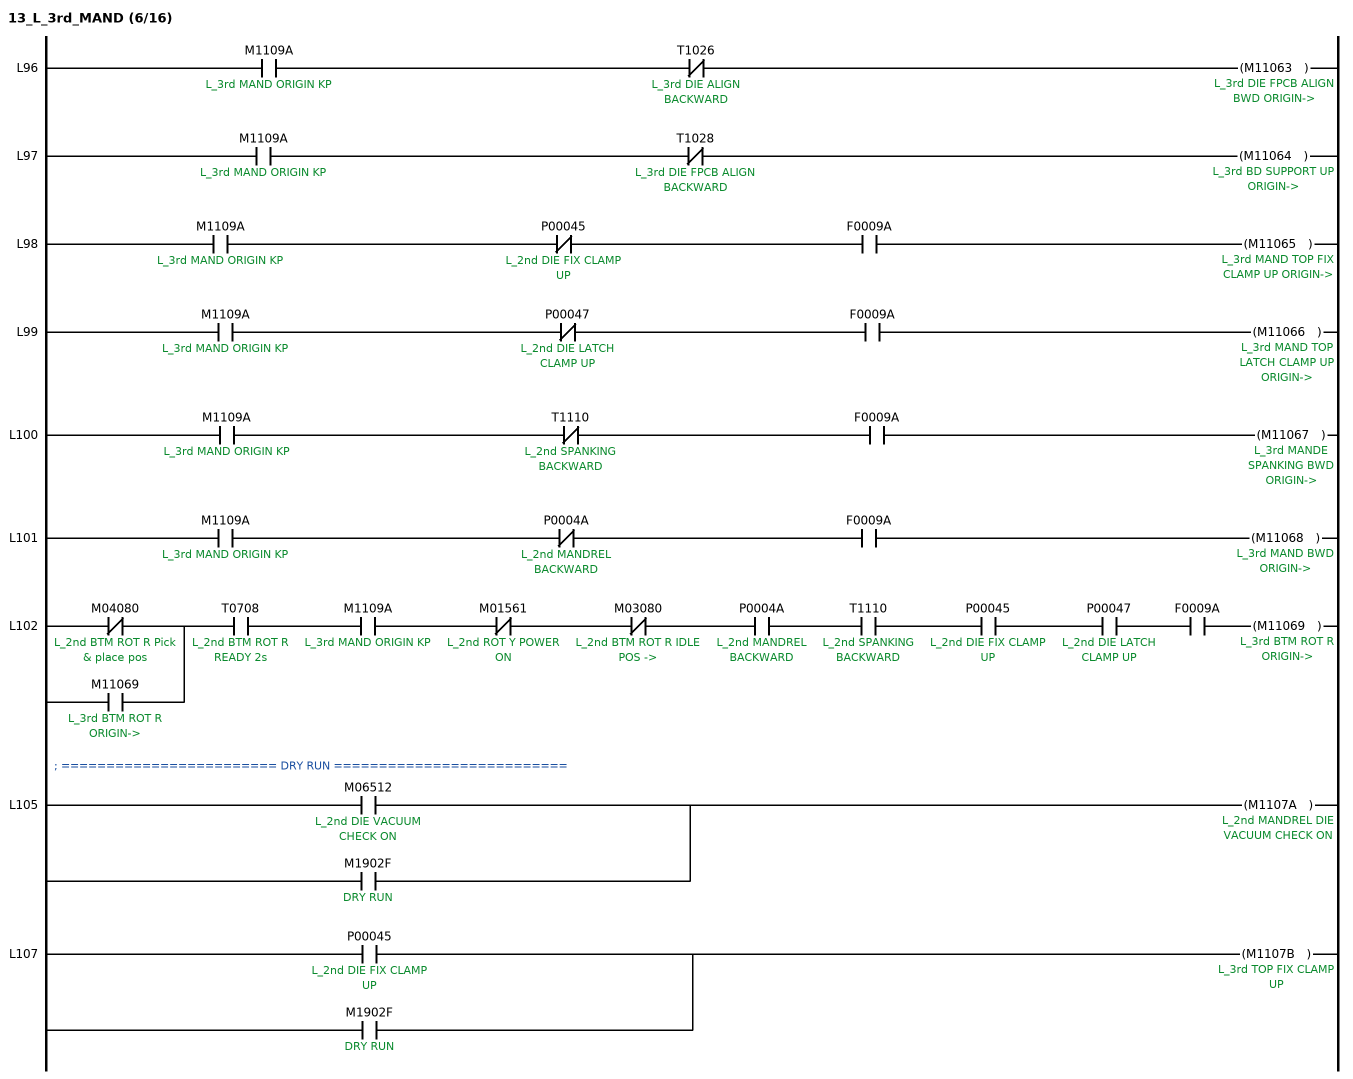
; L96
LOAD      M1109A	// L_3rd MAND ORIGIN KP
AND NOT   T1026	// L_3rd DIE ALIGN BACKWARD
OUT       M11063	// L_3rd DIE FPCB ALIGN BWD ORIGIN->
; L97
LOAD      M1109A	// L_3rd MAND ORIGIN KP
AND NOT   T1028	// L_3rd DIE FPCB ALIGN BACKWARD
OUT       M11064	// L_3rd BD SUPPORT UP ORIGIN->
; L98
LOAD      M1109A	// L_3rd MAND ORIGIN KP
AND NOT   P00045	// L_2nd DIE FIX CLAMP UP
AND       F0009A
OUT       M11065	// L_3rd MAND TOP FIX CLAMP UP ORIGIN->
; L99
LOAD      M1109A	// L_3rd MAND ORIGIN KP
AND NOT   P00047	// L_2nd DIE LATCH CLAMP UP
AND       F0009A
OUT       M11066	// L_3rd MAND TOP LATCH CLAMP UP ORIGIN->
; L100
LOAD      M1109A	// L_3rd MAND ORIGIN KP
AND NOT   T1110	// L_2nd SPANKING BACKWARD
AND       F0009A
OUT       M11067	// L_3rd MANDE SPANKING BWD ORIGIN->
; L101
LOAD      M1109A	// L_3rd MAND ORIGIN KP
AND NOT   P0004A	// L_2nd MANDREL BACKWARD
AND       F0009A
OUT       M11068	// L_3rd MAND BWD ORIGIN->
; L102
LOAD NOT  M04080	// L_2nd BTM ROT R Pick & place pos
OR        M11069	// L_3rd BTM ROT R ORIGIN->
AND       T0708	// L_2nd BTM ROT R READY 2s
AND       M1109A	// L_3rd MAND ORIGIN KP
AND NOT   M01561	// L_2nd ROT Y POWER ON
AND NOT   M03080	// L_2nd BTM ROT R IDLE POS ->
AND       P0004A	// L_2nd MANDREL BACKWARD
AND       T1110	// L_2nd SPANKING BACKWARD
AND       P00045	// L_2nd DIE FIX CLAMP UP
AND       P00047	// L_2nd DIE LATCH CLAMP UP
AND       F0009A
OUT       M11069	// L_3rd BTM ROT R ORIGIN->
// ======================== DRY RUN ==========================
; L105
LOAD      M06512	// L_2nd DIE VACUUM CHECK ON
OR        M1902F	// DRY RUN
OUT       M1107A	// L_2nd MANDREL DIE VACUUM CHECK ON
; L107
LOAD      P00045	// L_2nd DIE FIX CLAMP UP
OR        M1902F	// DRY RUN
OUT       M1107B	// L_3rd TOP FIX CLAMP UP

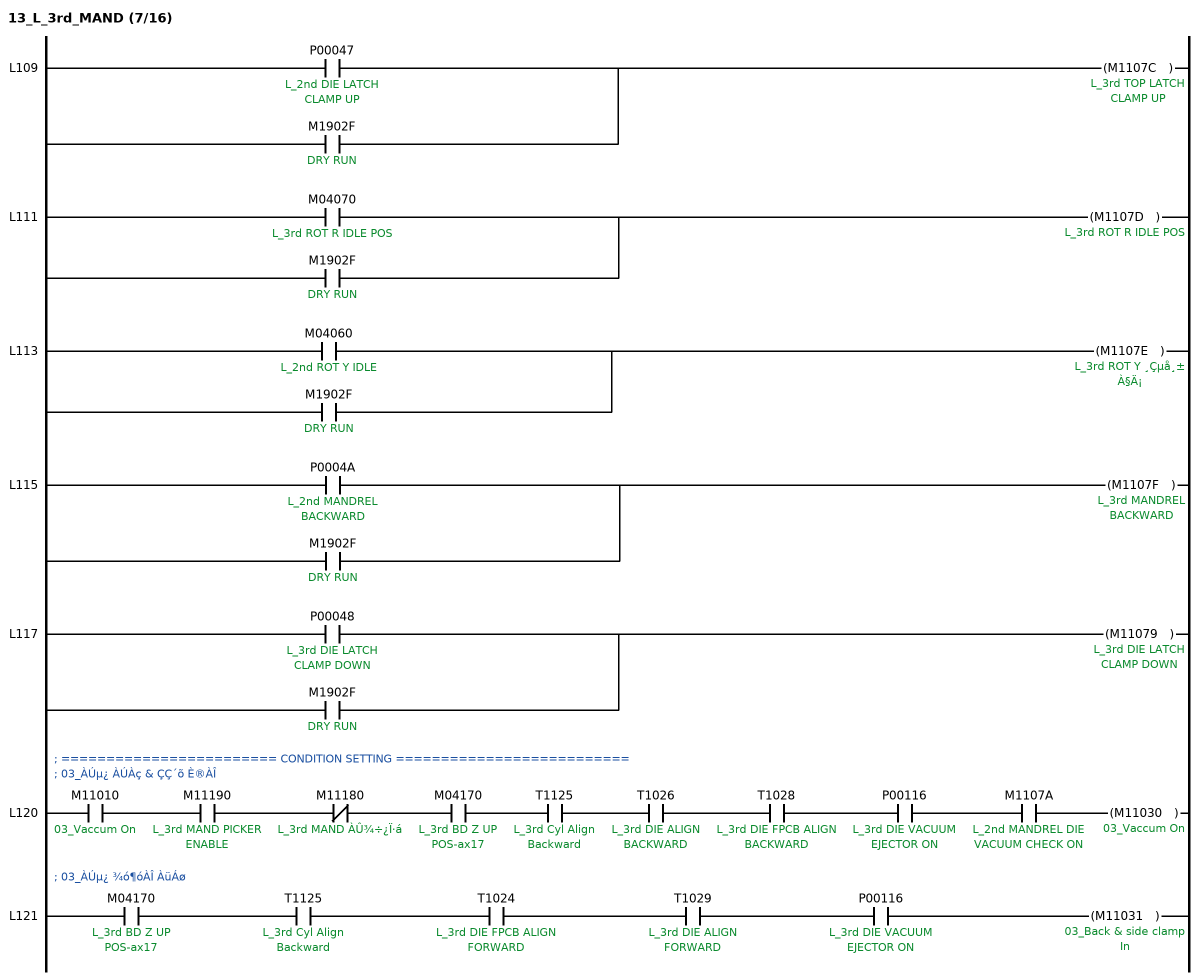
; L109
LOAD      P00047	// L_2nd DIE LATCH CLAMP UP
OR        M1902F	// DRY RUN
OUT       M1107C	// L_3rd TOP LATCH CLAMP UP
; L111
LOAD      M04070	// L_3rd ROT R IDLE POS
OR        M1902F	// DRY RUN
OUT       M1107D	// L_3rd ROT R IDLE POS
; L113
LOAD      M04060	// L_2nd ROT Y IDLE
OR        M1902F	// DRY RUN
OUT       M1107E	// L_3rd ROT Y ¸Çµå¸± À§Ä¡
; L115
LOAD      P0004A	// L_2nd MANDREL BACKWARD
OR        M1902F	// DRY RUN
OUT       M1107F	// L_3rd MANDREL BACKWARD
; L117
LOAD      P00048	// L_3rd DIE LATCH CLAMP DOWN
OR        M1902F	// DRY RUN
OUT       M11079	// L_3rd DIE LATCH CLAMP DOWN
// ======================== CONDITION SETTING ==========================
; L120
LOAD      M11010	// 03_Vaccum On
AND       M11190	// L_3rd MAND PICKER ENABLE
AND NOT   M11180	// L_3rd MAND ÀÛ¾÷¿Ï·á
AND       M04170	// L_3rd BD Z UP POS-ax17
AND       T1125	// L_3rd Cyl Align Backward
AND       T1026	// L_3rd DIE ALIGN BACKWARD
AND       T1028	// L_3rd DIE FPCB ALIGN BACKWARD
AND       P00116	// L_3rd DIE VACUUM EJECTOR ON
AND       M1107A	// L_2nd MANDREL DIE VACUUM CHECK ON
OUT       M11030	// 03_Vaccum On
// output comment: 03_ÀÚµ¿ ÀÚÀç & ÇÇ´õ È®ÀÎ
; L121
LOAD      M04170	// L_3rd BD Z UP POS-ax17
AND       T1125	// L_3rd Cyl Align Backward
AND       T1024	// L_3rd DIE FPCB ALIGN FORWARD
AND       T1029	// L_3rd DIE ALIGN FORWARD
AND       P00116	// L_3rd DIE VACUUM EJECTOR ON
OUT       M11031	// 03_Back & side clamp In
// output comment: 03_ÀÚµ¿ ¾ó¶óÀÎ ÀüÁø

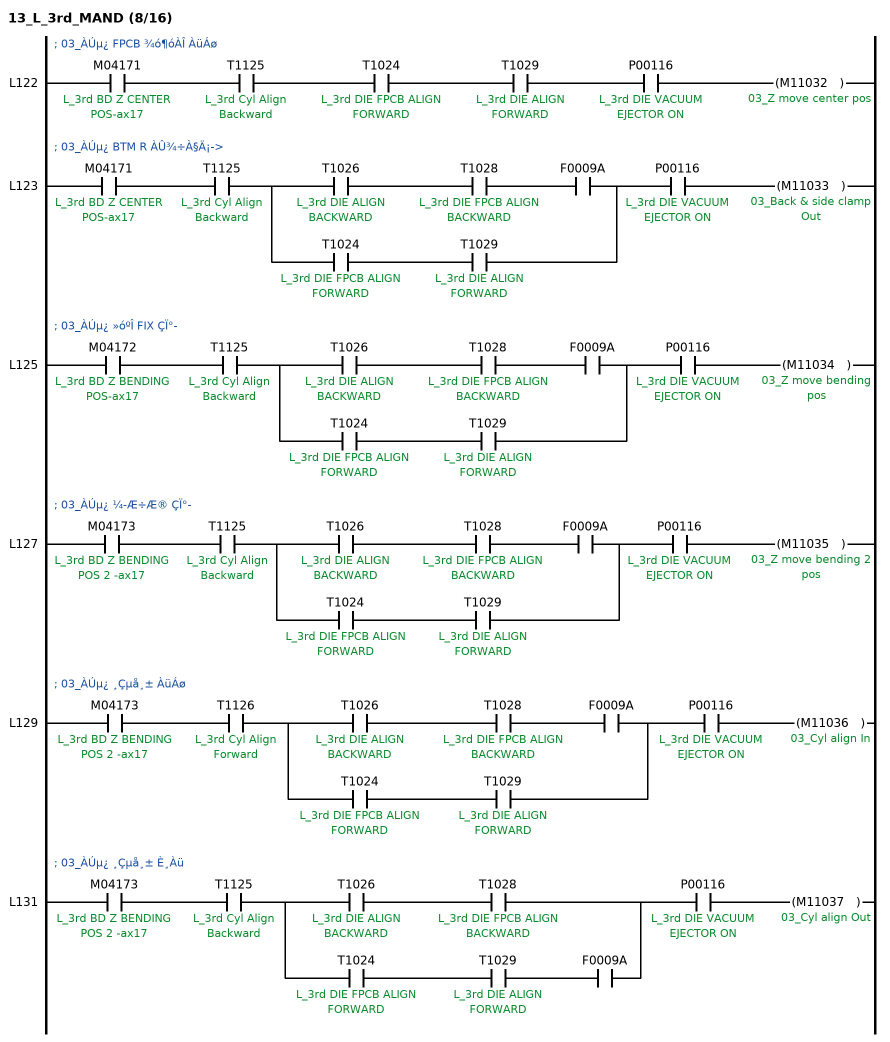
; L122
LOAD      M04171	// L_3rd BD Z CENTER POS-ax17
AND       T1125	// L_3rd Cyl Align Backward
AND       T1024	// L_3rd DIE FPCB ALIGN FORWARD
AND       T1029	// L_3rd DIE ALIGN FORWARD
AND       P00116	// L_3rd DIE VACUUM EJECTOR ON
OUT       M11032	// 03_Z move center pos
// output comment: 03_ÀÚµ¿ FPCB ¾ó¶óÀÎ ÀüÁø
; L123
LOAD      M04171	// L_3rd BD Z CENTER POS-ax17
AND       T1125	// L_3rd Cyl Align Backward
LOAD      T1026	// L_3rd DIE ALIGN BACKWARD
AND       T1028	// L_3rd DIE FPCB ALIGN BACKWARD
AND       F0009A
LOAD      T1024	// L_3rd DIE FPCB ALIGN FORWARD
AND       T1029	// L_3rd DIE ALIGN FORWARD
OR LOAD
AND LOAD
AND       P00116	// L_3rd DIE VACUUM EJECTOR ON
OUT       M11033	// 03_Back & side clamp Out
// output comment: 03_ÀÚµ¿ BTM R ÀÛ¾÷À§Ä¡->
; L125
LOAD      M04172	// L_3rd BD Z BENDING POS-ax17
AND       T1125	// L_3rd Cyl Align Backward
LOAD      T1026	// L_3rd DIE ALIGN BACKWARD
AND       T1028	// L_3rd DIE FPCB ALIGN BACKWARD
AND       F0009A
LOAD      T1024	// L_3rd DIE FPCB ALIGN FORWARD
AND       T1029	// L_3rd DIE ALIGN FORWARD
OR LOAD
AND LOAD
AND       P00116	// L_3rd DIE VACUUM EJECTOR ON
OUT       M11034	// 03_Z move bending pos
// output comment: 03_ÀÚµ¿ »óºÎ FIX ÇÏ°­
; L127
LOAD      M04173	// L_3rd BD Z BENDING POS 2 -ax17
AND       T1125	// L_3rd Cyl Align Backward
LOAD      T1026	// L_3rd DIE ALIGN BACKWARD
AND       T1028	// L_3rd DIE FPCB ALIGN BACKWARD
AND       F0009A
LOAD      T1024	// L_3rd DIE FPCB ALIGN FORWARD
AND       T1029	// L_3rd DIE ALIGN FORWARD
OR LOAD
AND LOAD
AND       P00116	// L_3rd DIE VACUUM EJECTOR ON
OUT       M11035	// 03_Z move bending 2 pos
// output comment: 03_ÀÚµ¿ ¼­Æ÷Æ® ÇÏ°­
; L129
LOAD      M04173	// L_3rd BD Z BENDING POS 2 -ax17
AND       T1126	// L_3rd Cyl Align Forward
LOAD      T1026	// L_3rd DIE ALIGN BACKWARD
AND       T1028	// L_3rd DIE FPCB ALIGN BACKWARD
AND       F0009A
LOAD      T1024	// L_3rd DIE FPCB ALIGN FORWARD
AND       T1029	// L_3rd DIE ALIGN FORWARD
OR LOAD
AND LOAD
AND       P00116	// L_3rd DIE VACUUM EJECTOR ON
OUT       M11036	// 03_Cyl align In
// output comment: 03_ÀÚµ¿ ¸Çµå¸± ÀüÁø
; L131
LOAD      M04173	// L_3rd BD Z BENDING POS 2 -ax17
AND       T1125	// L_3rd Cyl Align Backward
LOAD      T1026	// L_3rd DIE ALIGN BACKWARD
AND       T1028	// L_3rd DIE FPCB ALIGN BACKWARD
LOAD      T1024	// L_3rd DIE FPCB ALIGN FORWARD
AND       T1029	// L_3rd DIE ALIGN FORWARD
AND       F0009A
OR LOAD
AND LOAD
AND       P00116	// L_3rd DIE VACUUM EJECTOR ON
OUT       M11037	// 03_Cyl align Out
// output comment: 03_ÀÚµ¿ ¸Çµå¸± È¸Àü

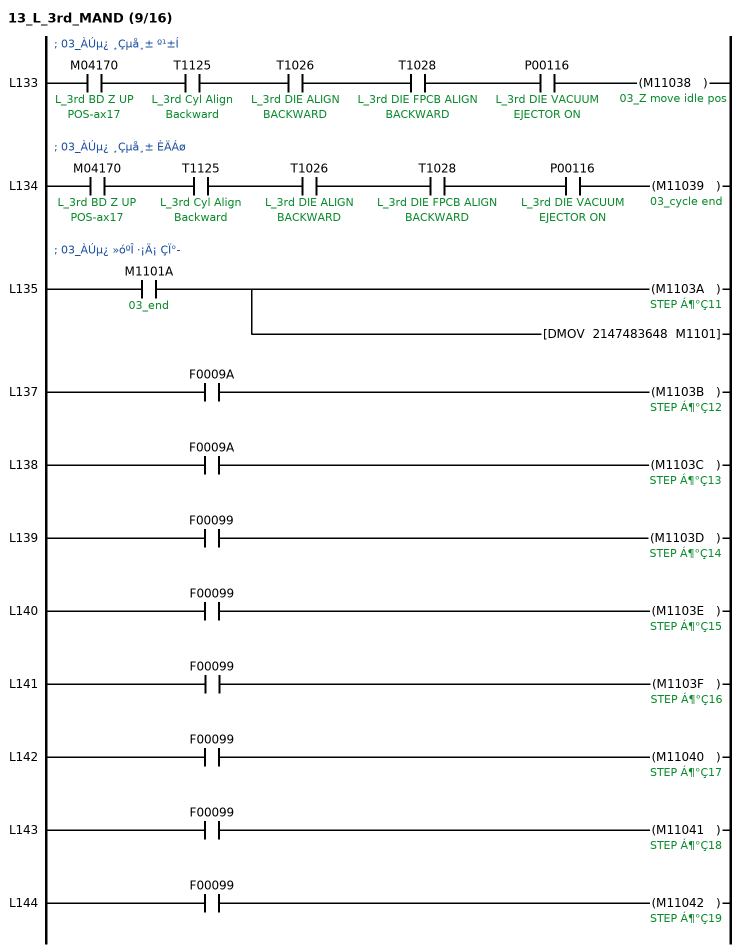
; L133
LOAD      M04170	// L_3rd BD Z UP POS-ax17
AND       T1125	// L_3rd Cyl Align Backward
AND       T1026	// L_3rd DIE ALIGN BACKWARD
AND       T1028	// L_3rd DIE FPCB ALIGN BACKWARD
AND       P00116	// L_3rd DIE VACUUM EJECTOR ON
OUT       M11038	// 03_Z move idle pos
// output comment: 03_ÀÚµ¿ ¸Çµå¸± º¹±Í
; L134
LOAD      M04170	// L_3rd BD Z UP POS-ax17
AND       T1125	// L_3rd Cyl Align Backward
AND       T1026	// L_3rd DIE ALIGN BACKWARD
AND       T1028	// L_3rd DIE FPCB ALIGN BACKWARD
AND       P00116	// L_3rd DIE VACUUM EJECTOR ON
OUT       M11039	// 03_cycle end
// output comment: 03_ÀÚµ¿ ¸Çµå¸± ÈÄÁø
; L135
LOAD      M1101A	// 03_end
OUT       M1103A	// STEP Á¶°Ç11
DMOV      2147483648 M1101
// output comment: 03_ÀÚµ¿ »óºÎ ·¡Ä¡ ÇÏ°­
; L137
LOAD      F0009A
OUT       M1103B	// STEP Á¶°Ç12
; L138
LOAD      F0009A
OUT       M1103C	// STEP Á¶°Ç13
; L139
LOAD      F00099
OUT       M1103D	// STEP Á¶°Ç14
; L140
LOAD      F00099
OUT       M1103E	// STEP Á¶°Ç15
; L141
LOAD      F00099
OUT       M1103F	// STEP Á¶°Ç16
; L142
LOAD      F00099
OUT       M11040	// STEP Á¶°Ç17
; L143
LOAD      F00099
OUT       M11041	// STEP Á¶°Ç18
; L144
LOAD      F00099
OUT       M11042	// STEP Á¶°Ç19

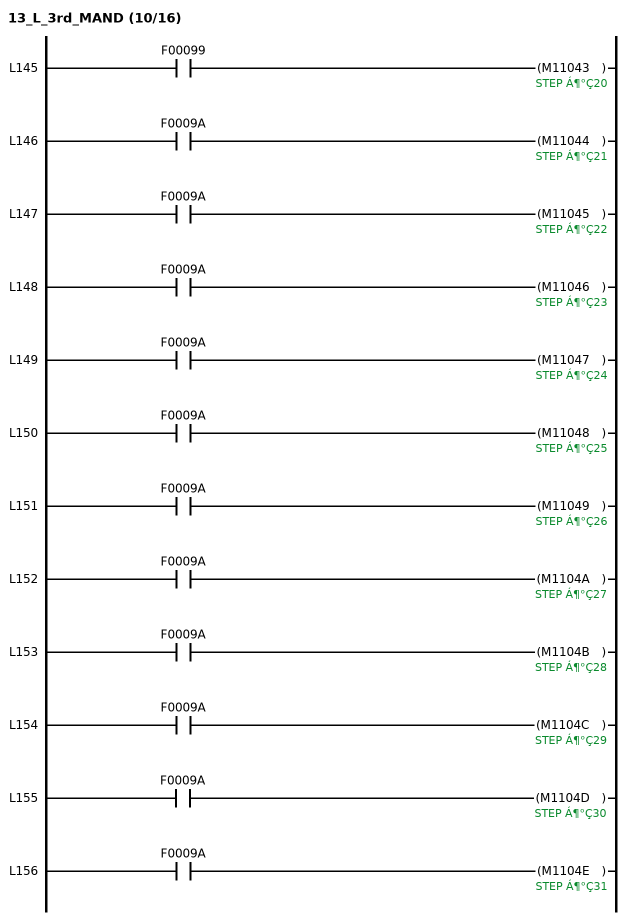
; L145
LOAD      F00099
OUT       M11043	// STEP Á¶°Ç20
; L146
LOAD      F0009A
OUT       M11044	// STEP Á¶°Ç21
; L147
LOAD      F0009A
OUT       M11045	// STEP Á¶°Ç22
; L148
LOAD      F0009A
OUT       M11046	// STEP Á¶°Ç23
; L149
LOAD      F0009A
OUT       M11047	// STEP Á¶°Ç24
; L150
LOAD      F0009A
OUT       M11048	// STEP Á¶°Ç25
; L151
LOAD      F0009A
OUT       M11049	// STEP Á¶°Ç26
; L152
LOAD      F0009A
OUT       M1104A	// STEP Á¶°Ç27
; L153
LOAD      F0009A
OUT       M1104B	// STEP Á¶°Ç28
; L154
LOAD      F0009A
OUT       M1104C	// STEP Á¶°Ç29
; L155
LOAD      F0009A
OUT       M1104D	// STEP Á¶°Ç30
; L156
LOAD      F0009A
OUT       M1104E	// STEP Á¶°Ç31

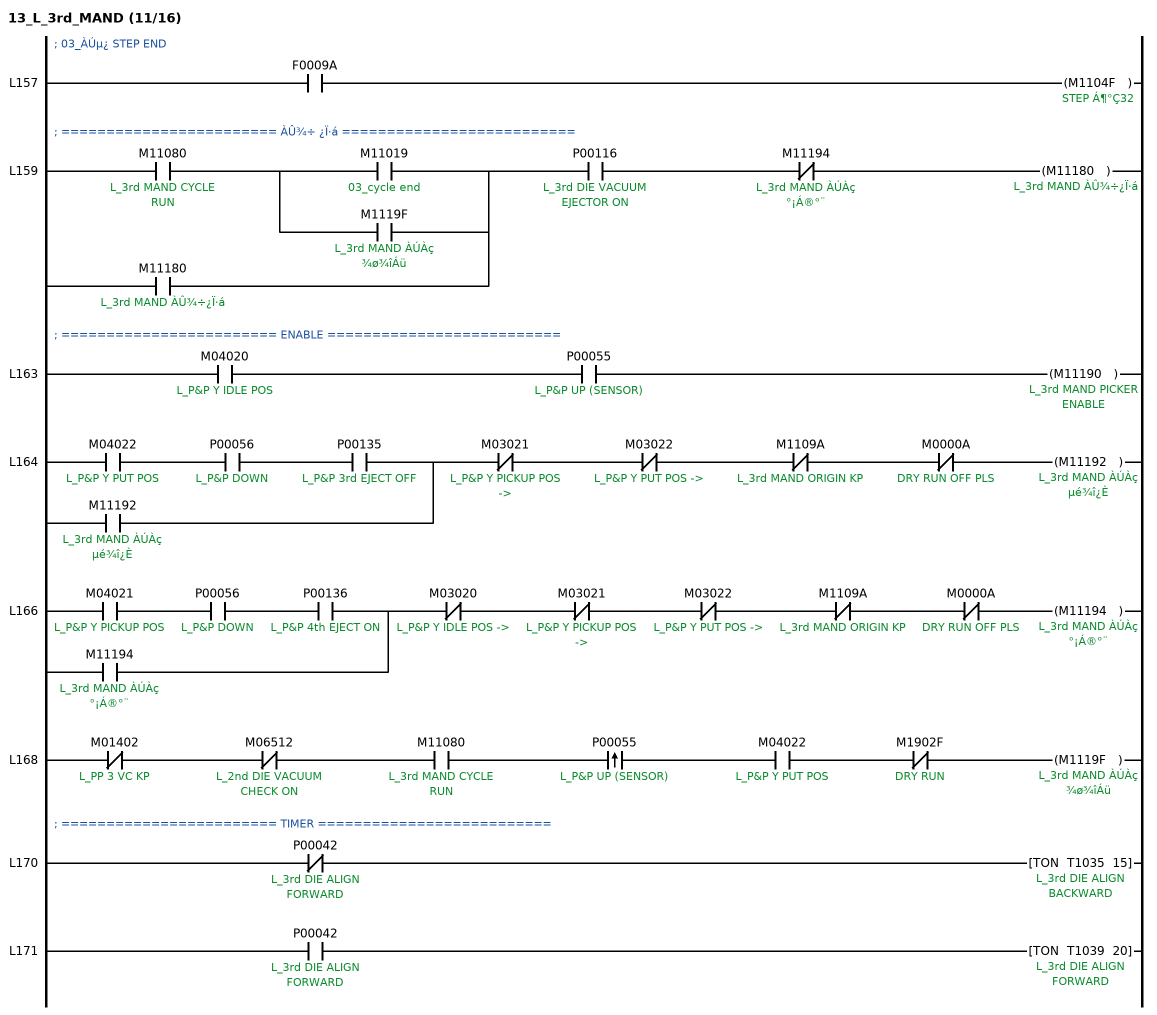
; L157
LOAD      F0009A
OUT       M1104F	// STEP Á¶°Ç32
// output comment: 03_ÀÚµ¿ STEP END
// ======================== ÀÛ¾÷ ¿Ï·á ==========================
; L159
LOAD      M11080	// L_3rd MAND CYCLE RUN
LOAD      M11019	// 03_cycle end
OR        M1119F	// L_3rd MAND ÀÚÀç ¾ø¾îÁü
AND LOAD
OR        M11180	// L_3rd MAND ÀÛ¾÷¿Ï·á
AND       P00116	// L_3rd DIE VACUUM EJECTOR ON
AND NOT   M11194	// L_3rd MAND ÀÚÀç °¡Á®°¨
OUT       M11180	// L_3rd MAND ÀÛ¾÷¿Ï·á
// ======================== ENABLE ==========================
; L163
LOAD      M04020	// L_P&P Y IDLE POS
AND       P00055	// L_P&P UP (SENSOR)
OUT       M11190	// L_3rd MAND PICKER ENABLE
; L164
LOAD      M04022	// L_P&P Y PUT POS
AND       P00056	// L_P&P DOWN
AND       P00135	// L_P&P 3rd EJECT OFF
OR        M11192	// L_3rd MAND ÀÚÀç µé¾î¿È
AND NOT   M03021	// L_P&P Y PICKUP POS ->
AND NOT   M03022	// L_P&P Y PUT POS ->
AND NOT   M1109A	// L_3rd MAND ORIGIN KP
AND NOT   M0000A	// DRY RUN OFF PLS
OUT       M11192	// L_3rd MAND ÀÚÀç µé¾î¿È
; L166
LOAD      M04021	// L_P&P Y PICKUP POS
AND       P00056	// L_P&P DOWN
AND       P00136	// L_P&P 4th EJECT ON
OR        M11194	// L_3rd MAND ÀÚÀç °¡Á®°¨
AND NOT   M03020	// L_P&P Y IDLE POS ->
AND NOT   M03021	// L_P&P Y PICKUP POS ->
AND NOT   M03022	// L_P&P Y PUT POS ->
AND NOT   M1109A	// L_3rd MAND ORIGIN KP
AND NOT   M0000A	// DRY RUN OFF PLS
OUT       M11194	// L_3rd MAND ÀÚÀç °¡Á®°¨
; L168
LOAD NOT  M01402	// L_PP 3 VC KP
AND NOT   M06512	// L_2nd DIE VACUUM CHECK ON
AND       M11080	// L_3rd MAND CYCLE RUN
ANDP      P00055	// L_P&P UP (SENSOR)
AND       M04022	// L_P&P Y PUT POS
AND NOT   M1902F	// DRY RUN
OUT       M1119F	// L_3rd MAND ÀÚÀç ¾ø¾îÁü
// ======================== TIMER ==========================
; L170
LOAD NOT  P00042	// L_3rd DIE ALIGN FORWARD
TON       T1035 15	// L_3rd DIE ALIGN BACKWARD
; L171
LOAD      P00042	// L_3rd DIE ALIGN FORWARD
TON       T1039 20	// L_3rd DIE ALIGN FORWARD

